ABB RAPID module: P90.mod

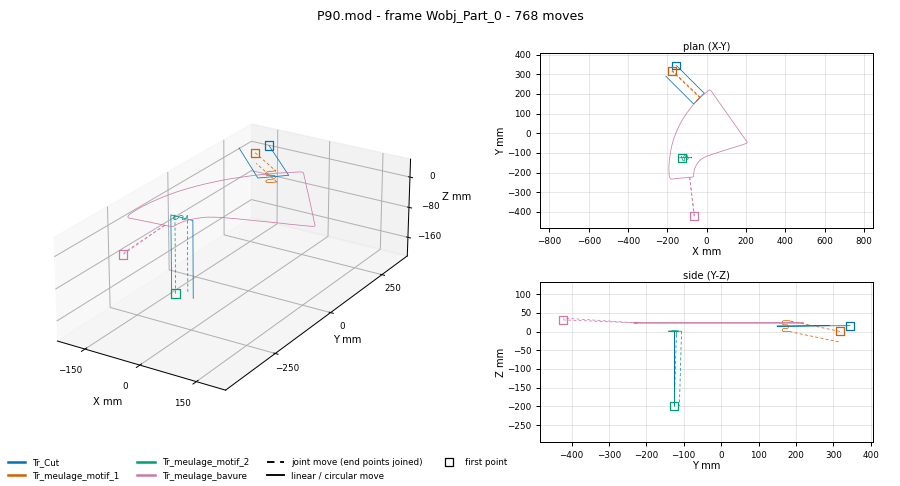
[picture p0: tool path of P90.mod in frame Wobj_Part_0, 768 of 778 moves have a stored position in this frame; points joined in program order, loops and branches not executed]
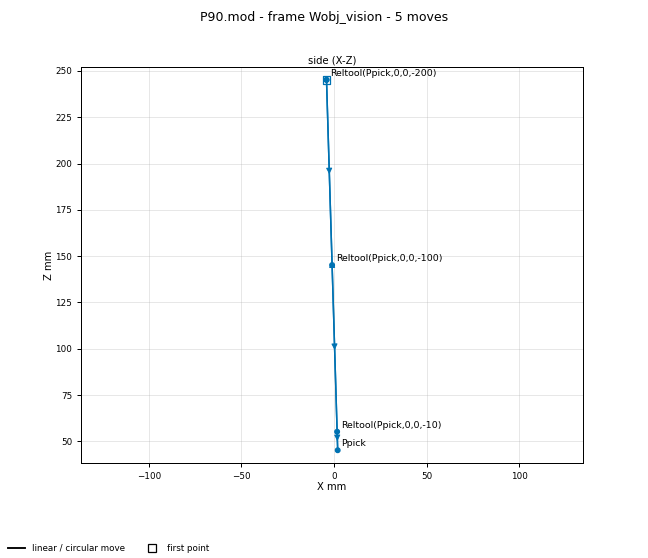
[picture p1: tool path of P90.mod in frame Wobj_vision, 5 of 778 moves have a stored position in this frame; points joined in program order, loops and branches not executed]
MODULE P90
	LOCAL CONST Speeddata vitesse_Tronconnage :=[10, 500, 0, 0];
	LOCAL CONST Robtarget Coupe_0 :=[[-42.54716015625,172.81159375,14.480369140625],[0.652659857981833,0.65438215651073,-0.267925350126422,-0.272093935579487],[0,0,0,0],[8.999999E+09,8.999999E+09,8.999999E+09,8.999999E+09,8.999999E+09,8.999999E+09]];
	LOCAL CONST Robtarget Coupe_1 :=[[-110.71790625,-124.2488046875,0.946675476074219],[0.708605063224334,-0.000599516120089683,-0.705604806156146,0.000602065284240644],[0,0,0,0],[8.999999E+09,8.999999E+09,8.999999E+09,8.999999E+09,8.999999E+09,8.999999E+09]];
	LOCAL CONST Robtarget Tr_meulage_motif_1_App1 :=[[-177.46862221102,317.614885440175,0.282455470844067],[0.29645362274748,-0.256571046125753,0.60201931555639,-0.695599950795604],[0,0,0,0],[8.999999E+09,8.999999E+09,8.999999E+09,8.999999E+09,8.999999E+09,8.999999E+09]];
	LOCAL CONST Robtarget Tr_meulage_motif_1_App2 :=[[-41.830808844926,187.387673178259,27.545191425886],[0.29645362274748,-0.256571046125753,0.60201931555639,-0.695599950795604],[0,0,0,0],[8.999999E+09,8.999999E+09,8.999999E+09,8.999999E+09,8.999999E+09,8.999999E+09]];
	LOCAL CONST Robtarget Tr_meulage_motif_1_P0 :=[[-34.6919765625,180.533609375,28.980072265625],[0.29645362274748,-0.256571046125753,0.60201931555639,-0.695599950795604],[0,0,0,0],[8.999999E+09,8.999999E+09,8.999999E+09,8.999999E+09,8.999999E+09,8.999999E+09]];
	LOCAL CONST Robtarget Tr_meulage_motif_1_P1 :=[[-35.39916796875,179.826578125,28.980072265625],[0.29645362274748,-0.256571046125753,0.60201931555639,-0.695599950795604],[0,0,0,0],[8.999999E+09,8.999999E+09,8.999999E+09,8.999999E+09,8.999999E+09,8.999999E+09]];
	LOCAL CONST Robtarget Tr_meulage_motif_1_P2 :=[[-36.106359375,179.1195625,28.980072265625],[0.29645362274748,-0.256571046125753,0.60201931555639,-0.695599950795604],[0,0,0,0],[8.999999E+09,8.999999E+09,8.999999E+09,8.999999E+09,8.999999E+09,8.999999E+09]];
	LOCAL CONST Robtarget Tr_meulage_motif_1_P3 :=[[-36.81355078125,178.41253125,28.980072265625],[0.29645362274748,-0.256571046125753,0.60201931555639,-0.695599950795604],[0,0,0,0],[8.999999E+09,8.999999E+09,8.999999E+09,8.999999E+09,8.999999E+09,8.999999E+09]];
	LOCAL CONST Robtarget Tr_meulage_motif_1_P4 :=[[-37.5207421875,177.705515625,28.980072265625],[0.29645362274748,-0.256571046125753,0.60201931555639,-0.695599950795604],[0,0,0,0],[8.999999E+09,8.999999E+09,8.999999E+09,8.999999E+09,8.999999E+09,8.999999E+09]];
	LOCAL CONST Robtarget Tr_meulage_motif_1_P5 :=[[-38.22793359375,176.9985,28.980072265625],[0.29645362274748,-0.256571046125753,0.60201931555639,-0.695599950795604],[0,0,0,0],[8.999999E+09,8.999999E+09,8.999999E+09,8.999999E+09,8.999999E+09,8.999999E+09]];
	LOCAL CONST Robtarget Tr_meulage_motif_1_P6 :=[[-38.935125,176.29146875,28.980072265625],[0.29645362274748,-0.256571046125753,0.60201931555639,-0.695599950795604],[0,0,0,0],[8.999999E+09,8.999999E+09,8.999999E+09,8.999999E+09,8.999999E+09,8.999999E+09]];
	LOCAL CONST Robtarget Tr_meulage_motif_1_P7 :=[[-39.64231640625,175.584453125,28.980072265625],[0.29645362274748,-0.256571046125753,0.60201931555639,-0.695599950795604],[0,0,0,0],[8.999999E+09,8.999999E+09,8.999999E+09,8.999999E+09,8.999999E+09,8.999999E+09]];
	LOCAL CONST Robtarget Tr_meulage_motif_1_P8 :=[[-40.3495078125,174.877421875,28.980072265625],[0.29645362274748,-0.256571046125753,0.60201931555639,-0.695599950795604],[0,0,0,0],[8.999999E+09,8.999999E+09,8.999999E+09,8.999999E+09,8.999999E+09,8.999999E+09]];
	LOCAL CONST Robtarget Tr_meulage_motif_1_P9 :=[[-41.05669921875,174.17040625,28.980072265625],[0.29645362274748,-0.256571046125753,0.60201931555639,-0.695599950795604],[0,0,0,0],[8.999999E+09,8.999999E+09,8.999999E+09,8.999999E+09,8.999999E+09,8.999999E+09]];
	LOCAL CONST Robtarget Tr_meulage_motif_1_P10 :=[[-41.76389453125,173.463390625,28.980072265625],[0.29645362274748,-0.256571046125753,0.60201931555639,-0.695599950795604],[0,0,0,0],[8.999999E+09,8.999999E+09,8.999999E+09,8.999999E+09,8.999999E+09,8.999999E+09]];
	LOCAL CONST Robtarget Tr_meulage_motif_1_P11 :=[[-42.4710859375,172.756359375,28.980072265625],[0.29645362274748,-0.256571046125753,0.60201931555639,-0.695599950795604],[0,0,0,0],[8.999999E+09,8.999999E+09,8.999999E+09,8.999999E+09,8.999999E+09,8.999999E+09]];
	LOCAL CONST Robtarget Tr_meulage_motif_1_P12 :=[[-43.17827734375,172.04934375,28.980072265625],[0.29645362274748,-0.256571046125753,0.60201931555639,-0.695599950795604],[0,0,0,0],[8.999999E+09,8.999999E+09,8.999999E+09,8.999999E+09,8.999999E+09,8.999999E+09]];
	LOCAL CONST Robtarget Tr_meulage_motif_1_P13 :=[[-43.88546875,171.3423125,28.980072265625],[0.29645362274748,-0.256571046125753,0.60201931555639,-0.695599950795604],[0,0,0,0],[8.999999E+09,8.999999E+09,8.999999E+09,8.999999E+09,8.999999E+09,8.999999E+09]];
	LOCAL CONST Robtarget Tr_meulage_motif_1_P14 :=[[-44.59266015625,170.635296875,28.980072265625],[0.29645362274748,-0.256571046125753,0.60201931555639,-0.695599950795604],[0,0,0,0],[8.999999E+09,8.999999E+09,8.999999E+09,8.999999E+09,8.999999E+09,8.999999E+09]];
	LOCAL CONST Robtarget Tr_meulage_motif_1_P15 :=[[-45.2998515625,169.92828125,28.980072265625],[0.29645362274748,-0.256571046125753,0.60201931555639,-0.695599950795604],[0,0,0,0],[8.999999E+09,8.999999E+09,8.999999E+09,8.999999E+09,8.999999E+09,8.999999E+09]];
	LOCAL CONST Robtarget Tr_meulage_motif_1_P16 :=[[-46.00704296875,169.22125,28.980072265625],[0.29645362274748,-0.256571046125753,0.60201931555639,-0.695599950795604],[0,0,0,0],[8.999999E+09,8.999999E+09,8.999999E+09,8.999999E+09,8.999999E+09,8.999999E+09]];
	LOCAL CONST Robtarget Tr_meulage_motif_1_P17 :=[[-46.714234375,168.514234375,28.980072265625],[0.29645362274748,-0.256571046125753,0.60201931555639,-0.695599950795604],[0,0,0,0],[8.999999E+09,8.999999E+09,8.999999E+09,8.999999E+09,8.999999E+09,8.999999E+09]];
	LOCAL CONST Robtarget Tr_meulage_motif_1_P18 :=[[-47.42142578125,167.807203125,28.980072265625],[0.29645362274748,-0.256571046125753,0.60201931555639,-0.695599950795604],[0,0,0,0],[8.999999E+09,8.999999E+09,8.999999E+09,8.999999E+09,8.999999E+09,8.999999E+09]];
	LOCAL CONST Robtarget Tr_meulage_motif_1_P19 :=[[-48.123859375,167.105953125,28.86948046875],[0.29645362274748,-0.256571046125753,0.60201931555639,-0.695599950795604],[0,0,0,0],[8.999999E+09,8.999999E+09,8.999999E+09,8.999999E+09,8.999999E+09,8.999999E+09]];
	LOCAL CONST Robtarget Tr_meulage_motif_1_P20 :=[[-48.794171875,166.437703125,28.658296875],[0.29645362274748,-0.256571046125753,0.60201931555639,-0.695599950795604],[0,0,0,0],[8.999999E+09,8.999999E+09,8.999999E+09,8.999999E+09,8.999999E+09,8.999999E+09]];
	LOCAL CONST Robtarget Tr_meulage_motif_1_P21 :=[[-49.3984375,165.836046875,28.386458984375],[0.29645362274748,-0.256571046125753,0.60201931555639,-0.695599950795604],[0,0,0,0],[8.999999E+09,8.999999E+09,8.999999E+09,8.999999E+09,8.999999E+09,8.999999E+09]];
	LOCAL CONST Robtarget Tr_meulage_motif_1_P22 :=[[-49.9300390625,165.307078125,28.11052734375],[0.29645362274748,-0.256571046125753,0.60201931555639,-0.695599950795604],[0,0,0,0],[8.999999E+09,8.999999E+09,8.999999E+09,8.999999E+09,8.999999E+09,8.999999E+09]];
	LOCAL CONST Robtarget Tr_meulage_motif_1_P23 :=[[-50.71148828125,164.531390625,27.494416015625],[0.29645362274748,-0.256571046125753,0.60201931555639,-0.695599950795604],[0,0,0,0],[8.999999E+09,8.999999E+09,8.999999E+09,8.999999E+09,8.999999E+09,8.999999E+09]];
	LOCAL CONST Robtarget Tr_meulage_motif_1_P24 :=[[-51.43940234375,163.811328125,26.64677734375],[0.29645362274748,-0.256571046125753,0.60201931555639,-0.695599950795604],[0,0,0,0],[8.999999E+09,8.999999E+09,8.999999E+09,8.999999E+09,8.999999E+09,8.999999E+09]];
	LOCAL CONST Robtarget Tr_meulage_motif_1_P25 :=[[-52.04349609375,163.21665625,25.622921875],[0.29645362274748,-0.256571046125753,0.60201931555639,-0.695599950795604],[0,0,0,0],[8.999999E+09,8.999999E+09,8.999999E+09,8.999999E+09,8.999999E+09,8.999999E+09]];
	LOCAL CONST Robtarget Tr_meulage_motif_1_P26 :=[[-52.393765625,162.8765625,24.5067578125],[0.29645362274748,-0.256571046125753,0.60201931555639,-0.695599950795604],[0,0,0,0],[8.999999E+09,8.999999E+09,8.999999E+09,8.999999E+09,8.999999E+09,8.999999E+09]];
	LOCAL CONST Robtarget Tr_meulage_motif_1_P27 :=[[-52.41605859375,162.86059375,23.810802734375],[0.29645362274748,-0.256571046125753,0.60201931555639,-0.695599950795604],[0,0,0,0],[8.999999E+09,8.999999E+09,8.999999E+09,8.999999E+09,8.999999E+09,8.999999E+09]];
	LOCAL CONST Robtarget Tr_meulage_motif_1_P28 :=[[-52.41905078125,162.863578125,23.14956640625],[0.29645362274748,-0.256571046125753,0.60201931555639,-0.695599950795604],[0,0,0,0],[8.999999E+09,8.999999E+09,8.999999E+09,8.999999E+09,8.999999E+09,8.999999E+09]];
	LOCAL CONST Robtarget Tr_meulage_motif_1_P29 :=[[-52.383234375,162.905375,22.488486328125],[0.29645362274748,-0.256571046125753,0.60201931555639,-0.695599950795604],[0,0,0,0],[8.999999E+09,8.999999E+09,8.999999E+09,8.999999E+09,8.999999E+09,8.999999E+09]];
	LOCAL CONST Robtarget Tr_meulage_motif_1_P30 :=[[-52.03588671875,163.262609375,21.386759765625],[0.29645362274748,-0.256571046125753,0.60201931555639,-0.695599950795604],[0,0,0,0],[8.999999E+09,8.999999E+09,8.999999E+09,8.999999E+09,8.999999E+09,8.999999E+09]];
	LOCAL CONST Robtarget Tr_meulage_motif_1_P31 :=[[-51.4346484375,163.872828125,20.380154296875],[0.29645362274748,-0.256571046125753,0.60201931555639,-0.695599950795604],[0,0,0,0],[8.999999E+09,8.999999E+09,8.999999E+09,8.999999E+09,8.999999E+09,8.999999E+09]];
	LOCAL CONST Robtarget Tr_meulage_motif_1_P32 :=[[-50.71465625,164.600140625,19.551296875],[0.29645362274748,-0.256571046125753,0.60201931555639,-0.695599950795604],[0,0,0,0],[8.999999E+09,8.999999E+09,8.999999E+09,8.999999E+09,8.999999E+09,8.999999E+09]];
	LOCAL CONST Robtarget Tr_meulage_motif_1_P33 :=[[-50.2305390625,165.087734375,19.1555546875],[0.29645362274748,-0.256571046125753,0.60201931555639,-0.695599950795604],[0,0,0,0],[8.999999E+09,8.999999E+09,8.999999E+09,8.999999E+09,8.999999E+09,8.999999E+09]];
	LOCAL CONST Robtarget Tr_meulage_motif_1_P34 :=[[-49.41370703125,165.90878125,18.668033203125],[0.29645362274748,-0.256571046125753,0.60201931555639,-0.695599950795604],[0,0,0,0],[8.999999E+09,8.999999E+09,8.999999E+09,8.999999E+09,8.999999E+09,8.999999E+09]];
	LOCAL CONST Robtarget Tr_meulage_motif_1_P35 :=[[-48.8173046875,166.5074375,18.4039453125],[0.29645362274748,-0.256571046125753,0.60201931555639,-0.695599950795604],[0,0,0,0],[8.999999E+09,8.999999E+09,8.999999E+09,8.999999E+09,8.999999E+09,8.999999E+09]];
	LOCAL CONST Robtarget Tr_meulage_motif_1_P36 :=[[-48.15912890625,167.167296875,18.19948046875],[0.29645362274748,-0.256571046125753,0.60201931555639,-0.695599950795604],[0,0,0,0],[8.999999E+09,8.999999E+09,8.999999E+09,8.999999E+09,8.999999E+09,8.999999E+09]];
	LOCAL CONST Robtarget Tr_meulage_motif_1_P37 :=[[-47.46546484375,167.86178125,18.090888671875],[0.29645362274748,-0.256571046125753,0.60201931555639,-0.695599950795604],[0,0,0,0],[8.999999E+09,8.999999E+09,8.999999E+09,8.999999E+09,8.999999E+09,8.999999E+09]];
	LOCAL CONST Robtarget Tr_meulage_motif_1_P38 :=[[-46.76403515625,168.564046875,17.980296875],[0.29645362274748,-0.256571046125753,0.60201931555639,-0.695599950795604],[0,0,0,0],[8.999999E+09,8.999999E+09,8.999999E+09,8.999999E+09,8.999999E+09,8.999999E+09]];
	LOCAL CONST Robtarget Tr_meulage_motif_1_P39 :=[[-46.05684375,169.2710625,17.980296875],[0.29645362274748,-0.256571046125753,0.60201931555639,-0.695599950795604],[0,0,0,0],[8.999999E+09,8.999999E+09,8.999999E+09,8.999999E+09,8.999999E+09,8.999999E+09]];
	LOCAL CONST Robtarget Tr_meulage_motif_1_P40 :=[[-45.34965234375,169.97809375,17.980296875],[0.29645362274748,-0.256571046125753,0.60201931555639,-0.695599950795604],[0,0,0,0],[8.999999E+09,8.999999E+09,8.999999E+09,8.999999E+09,8.999999E+09,8.999999E+09]];
	LOCAL CONST Robtarget Tr_meulage_motif_1_P41 :=[[-44.6424609375,170.685109375,17.980296875],[0.29645362274748,-0.256571046125753,0.60201931555639,-0.695599950795604],[0,0,0,0],[8.999999E+09,8.999999E+09,8.999999E+09,8.999999E+09,8.999999E+09,8.999999E+09]];
	LOCAL CONST Robtarget Tr_meulage_motif_1_P42 :=[[-43.935265625,171.392125,17.980296875],[0.29645362274748,-0.256571046125753,0.60201931555639,-0.695599950795604],[0,0,0,0],[8.999999E+09,8.999999E+09,8.999999E+09,8.999999E+09,8.999999E+09,8.999999E+09]];
	LOCAL CONST Robtarget Tr_meulage_motif_1_P43 :=[[-43.22807421875,172.09915625,17.980296875],[0.29645362274748,-0.256571046125753,0.60201931555639,-0.695599950795604],[0,0,0,0],[8.999999E+09,8.999999E+09,8.999999E+09,8.999999E+09,8.999999E+09,8.999999E+09]];
	LOCAL CONST Robtarget Tr_meulage_motif_1_P44 :=[[-42.5208828125,172.806171875,17.980296875],[0.29645362274748,-0.256571046125753,0.60201931555639,-0.695599950795604],[0,0,0,0],[8.999999E+09,8.999999E+09,8.999999E+09,8.999999E+09,8.999999E+09,8.999999E+09]];
	LOCAL CONST Robtarget Tr_meulage_motif_1_P45 :=[[-41.81369140625,173.5131875,17.980296875],[0.29645362274748,-0.256571046125753,0.60201931555639,-0.695599950795604],[0,0,0,0],[8.999999E+09,8.999999E+09,8.999999E+09,8.999999E+09,8.999999E+09,8.999999E+09]];
	LOCAL CONST Robtarget Tr_meulage_motif_1_P46 :=[[-41.1065,174.22021875,17.980296875],[0.29645362274748,-0.256571046125753,0.60201931555639,-0.695599950795604],[0,0,0,0],[8.999999E+09,8.999999E+09,8.999999E+09,8.999999E+09,8.999999E+09,8.999999E+09]];
	LOCAL CONST Robtarget Tr_meulage_motif_1_P47 :=[[-40.39930859375,174.927234375,17.980296875],[0.29645362274748,-0.256571046125753,0.60201931555639,-0.695599950795604],[0,0,0,0],[8.999999E+09,8.999999E+09,8.999999E+09,8.999999E+09,8.999999E+09,8.999999E+09]];
	LOCAL CONST Robtarget Tr_meulage_motif_1_P48 :=[[-39.6921171875,175.634265625,17.980296875],[0.29645362274748,-0.256571046125753,0.60201931555639,-0.695599950795604],[0,0,0,0],[8.999999E+09,8.999999E+09,8.999999E+09,8.999999E+09,8.999999E+09,8.999999E+09]];
	LOCAL CONST Robtarget Tr_meulage_motif_1_P49 :=[[-38.99068359375,176.33653125,17.869705078125],[0.29645362274748,-0.256571046125753,0.60201931555639,-0.695599950795604],[0,0,0,0],[8.999999E+09,8.999999E+09,8.999999E+09,8.999999E+09,8.999999E+09,8.999999E+09]];
	LOCAL CONST Robtarget Tr_meulage_motif_1_P50 :=[[-38.32228515625,177.006671875,17.6585234375],[0.29645362274748,-0.256571046125753,0.60201931555639,-0.695599950795604],[0,0,0,0],[8.999999E+09,8.999999E+09,8.999999E+09,8.999999E+09,8.999999E+09,8.999999E+09]];
	LOCAL CONST Robtarget Tr_meulage_motif_1_P51 :=[[-37.72048046875,177.610796875,17.38668359375],[0.29645362274748,-0.256571046125753,0.60201931555639,-0.695599950795604],[0,0,0,0],[8.999999E+09,8.999999E+09,8.999999E+09,8.999999E+09,8.999999E+09,8.999999E+09]];
	LOCAL CONST Robtarget Tr_meulage_motif_1_P52 :=[[-37.2186875,178.11521875,17.08253515625],[0.29645362274748,-0.256571046125753,0.60201931555639,-0.695599950795604],[0,0,0,0],[8.999999E+09,8.999999E+09,8.999999E+09,8.999999E+09,8.999999E+09,8.999999E+09]];
	LOCAL CONST Robtarget Tr_meulage_motif_1_P53 :=[[-36.49012109375,178.849609375,16.420015625],[0.29645362274748,-0.256571046125753,0.60201931555639,-0.695599950795604],[0,0,0,0],[8.999999E+09,8.999999E+09,8.999999E+09,8.999999E+09,8.999999E+09,8.999999E+09]];
	LOCAL CONST Robtarget Tr_meulage_motif_1_P54 :=[[-35.85636328125,179.491390625,15.51809765625],[0.29645362274748,-0.256571046125753,0.60201931555639,-0.695599950795604],[0,0,0,0],[8.999999E+09,8.999999E+09,8.999999E+09,8.999999E+09,8.999999E+09,8.999999E+09]];
	LOCAL CONST Robtarget Tr_meulage_motif_1_P55 :=[[-35.4827734375,179.874359375,14.472087890625],[0.29645362274748,-0.256571046125753,0.60201931555639,-0.695599950795604],[0,0,0,0],[8.999999E+09,8.999999E+09,8.999999E+09,8.999999E+09,8.999999E+09,8.999999E+09]];
	LOCAL CONST Robtarget Tr_meulage_motif_1_P56 :=[[-35.355234375,180.008140625,13.7788828125],[0.29645362274748,-0.256571046125753,0.60201931555639,-0.695599950795604],[0,0,0,0],[8.999999E+09,8.999999E+09,8.999999E+09,8.999999E+09,8.999999E+09,8.999999E+09]];
	LOCAL CONST Robtarget Tr_meulage_motif_1_P57 :=[[-35.3135703125,180.056765625,13.0088984375],[0.29645362274748,-0.256571046125753,0.60201931555639,-0.695599950795604],[0,0,0,0],[8.999999E+09,8.999999E+09,8.999999E+09,8.999999E+09,8.999999E+09,8.999999E+09]];
	LOCAL CONST Robtarget Tr_meulage_motif_1_P58 :=[[-35.36439453125,180.012921875,12.2390400390625],[0.29645362274748,-0.256571046125753,0.60201931555639,-0.695599950795604],[0,0,0,0],[8.999999E+09,8.999999E+09,8.999999E+09,8.999999E+09,8.999999E+09,8.999999E+09]];
	LOCAL CONST Robtarget Tr_meulage_motif_1_P59 :=[[-35.66614453125,179.72128125,11.1308125],[0.29645362274748,-0.256571046125753,0.60201931555639,-0.695599950795604],[0,0,0,0],[8.999999E+09,8.999999E+09,8.999999E+09,8.999999E+09,8.999999E+09,8.999999E+09]];
	LOCAL CONST Robtarget Tr_meulage_motif_1_P60 :=[[-35.96179296875,179.431015625,10.54513671875],[0.29645362274748,-0.256571046125753,0.60201931555639,-0.695599950795604],[0,0,0,0],[8.999999E+09,8.999999E+09,8.999999E+09,8.999999E+09,8.999999E+09,8.999999E+09]];
	LOCAL CONST Robtarget Tr_meulage_motif_1_P61 :=[[-36.59317578125,178.8078125,9.6580302734375],[0.29645362274748,-0.256571046125753,0.60201931555639,-0.695599950795604],[0,0,0,0],[8.999999E+09,8.999999E+09,8.999999E+09,8.999999E+09,8.999999E+09,8.999999E+09]];
	LOCAL CONST Robtarget Tr_meulage_motif_1_P62 :=[[-37.00924609375,178.39559375,9.2437265625],[0.29645362274748,-0.256571046125753,0.60201931555639,-0.695599950795604],[0,0,0,0],[8.999999E+09,8.999999E+09,8.999999E+09,8.999999E+09,8.999999E+09,8.999999E+09]];
	LOCAL CONST Robtarget Tr_meulage_motif_1_P63 :=[[-37.80228515625,177.607671875,8.6996435546875],[0.29645362274748,-0.256571046125753,0.60201931555639,-0.695599950795604],[0,0,0,0],[8.999999E+09,8.999999E+09,8.999999E+09,8.999999E+09,8.999999E+09,8.999999E+09]];
	LOCAL CONST Robtarget Tr_meulage_motif_1_P64 :=[[-38.3874765625,177.025296875,8.4041494140625],[0.29645362274748,-0.256571046125753,0.60201931555639,-0.695599950795604],[0,0,0,0],[8.999999E+09,8.999999E+09,8.999999E+09,8.999999E+09,8.999999E+09,8.999999E+09]];
	LOCAL CONST Robtarget Tr_meulage_motif_1_P65 :=[[-39.04750390625,176.36728125,8.199685546875],[0.29645362274748,-0.256571046125753,0.60201931555639,-0.695599950795604],[0,0,0,0],[8.999999E+09,8.999999E+09,8.999999E+09,8.999999E+09,8.999999E+09,8.999999E+09]];
	LOCAL CONST Robtarget Tr_meulage_motif_1_P66 :=[[-39.7421484375,175.67378125,8.09109375],[0.29645362274748,-0.256571046125753,0.60201931555639,-0.695599950795604],[0,0,0,0],[8.999999E+09,8.999999E+09,8.999999E+09,8.999999E+09,8.999999E+09,8.999999E+09]];
	LOCAL CONST Robtarget Tr_meulage_motif_1_P67 :=[[-40.44458203125,174.972515625,7.98050244140625],[0.29645362274748,-0.256571046125753,0.60201931555639,-0.695599950795604],[0,0,0,0],[8.999999E+09,8.999999E+09,8.999999E+09,8.999999E+09,8.999999E+09,8.999999E+09]];
	LOCAL CONST Robtarget Tr_meulage_motif_1_P68 :=[[-41.1517734375,174.2655,7.98050244140625],[0.29645362274748,-0.256571046125753,0.60201931555639,-0.695599950795604],[0,0,0,0],[8.999999E+09,8.999999E+09,8.999999E+09,8.999999E+09,8.999999E+09,8.999999E+09]];
	LOCAL CONST Robtarget Tr_meulage_motif_1_P69 :=[[-41.85896484375,173.558484375,7.98050244140625],[0.29645362274748,-0.256571046125753,0.60201931555639,-0.695599950795604],[0,0,0,0],[8.999999E+09,8.999999E+09,8.999999E+09,8.999999E+09,8.999999E+09,8.999999E+09]];
	LOCAL CONST Robtarget Tr_meulage_motif_1_P70 :=[[-42.56615625,172.851453125,7.98050244140625],[0.29645362274748,-0.256571046125753,0.60201931555639,-0.695599950795604],[0,0,0,0],[8.999999E+09,8.999999E+09,8.999999E+09,8.999999E+09,8.999999E+09,8.999999E+09]];
	LOCAL CONST Robtarget Tr_meulage_motif_1_P71 :=[[-43.27334765625,172.1444375,7.98050244140625],[0.29645362274748,-0.256571046125753,0.60201931555639,-0.695599950795604],[0,0,0,0],[8.999999E+09,8.999999E+09,8.999999E+09,8.999999E+09,8.999999E+09,8.999999E+09]];
	LOCAL CONST Robtarget Tr_meulage_motif_1_P72 :=[[-43.9805390625,171.43740625,7.98050244140625],[0.29645362274748,-0.256571046125753,0.60201931555639,-0.695599950795604],[0,0,0,0],[8.999999E+09,8.999999E+09,8.999999E+09,8.999999E+09,8.999999E+09,8.999999E+09]];
	LOCAL CONST Robtarget Tr_meulage_motif_1_P73 :=[[-44.68773046875,170.730390625,7.98050244140625],[0.29645362274748,-0.256571046125753,0.60201931555639,-0.695599950795604],[0,0,0,0],[8.999999E+09,8.999999E+09,8.999999E+09,8.999999E+09,8.999999E+09,8.999999E+09]];
	LOCAL CONST Robtarget Tr_meulage_motif_1_P74 :=[[-45.394921875,170.023375,7.98050244140625],[0.29645362274748,-0.256571046125753,0.60201931555639,-0.695599950795604],[0,0,0,0],[8.999999E+09,8.999999E+09,8.999999E+09,8.999999E+09,8.999999E+09,8.999999E+09]];
	LOCAL CONST Robtarget Tr_meulage_motif_1_P75 :=[[-46.10211328125,169.31634375,7.98050244140625],[0.29645362274748,-0.256571046125753,0.60201931555639,-0.695599950795604],[0,0,0,0],[8.999999E+09,8.999999E+09,8.999999E+09,8.999999E+09,8.999999E+09,8.999999E+09]];
	LOCAL CONST Robtarget Tr_meulage_motif_1_P76 :=[[-46.80930859375,168.609328125,7.98050244140625],[0.29645362274748,-0.256571046125753,0.60201931555639,-0.695599950795604],[0,0,0,0],[8.999999E+09,8.999999E+09,8.999999E+09,8.999999E+09,8.999999E+09,8.999999E+09]];
	LOCAL CONST Robtarget Tr_meulage_motif_1_P77 :=[[-47.5165,167.902296875,7.9805029296875],[0.29645362274748,-0.256571046125753,0.60201931555639,-0.695599950795604],[0,0,0,0],[8.999999E+09,8.999999E+09,8.999999E+09,8.999999E+09,8.999999E+09,8.999999E+09]];
	LOCAL CONST Robtarget Tr_meulage_motif_1_P78 :=[[-48.2189296875,167.201046875,7.8699111328125],[0.29645362274748,-0.256571046125753,0.60201931555639,-0.695599950795604],[0,0,0,0],[8.999999E+09,8.999999E+09,8.999999E+09,8.999999E+09,8.999999E+09,8.999999E+09]];
	LOCAL CONST Robtarget Tr_meulage_motif_1_P79 :=[[-48.88924609375,166.532796875,7.65872802734375],[0.29645362274748,-0.256571046125753,0.60201931555639,-0.695599950795604],[0,0,0,0],[8.999999E+09,8.999999E+09,8.999999E+09,8.999999E+09,8.999999E+09,8.999999E+09]];
	LOCAL CONST Robtarget Tr_meulage_motif_1_P80 :=[[-49.49351171875,165.931140625,7.38689013671875],[0.29645362274748,-0.256571046125753,0.60201931555639,-0.695599950795604],[0,0,0,0],[8.999999E+09,8.999999E+09,8.999999E+09,8.999999E+09,8.999999E+09,8.999999E+09]];
	LOCAL CONST Robtarget Tr_meulage_motif_1_P81 :=[[-50.025109375,165.402171875,7.1109580078125],[0.29645362274748,-0.256571046125753,0.60201931555639,-0.695599950795604],[0,0,0,0],[8.999999E+09,8.999999E+09,8.999999E+09,8.999999E+09,8.999999E+09,8.999999E+09]];
	LOCAL CONST Robtarget Tr_meulage_motif_1_P82 :=[[-50.8065625,164.626484375,6.494845703125],[0.29645362274748,-0.256571046125753,0.60201931555639,-0.695599950795604],[0,0,0,0],[8.999999E+09,8.999999E+09,8.999999E+09,8.999999E+09,8.999999E+09,8.999999E+09]];
	LOCAL CONST Robtarget Tr_meulage_motif_1_P83 :=[[-51.48719140625,163.954109375,5.6008955078125],[0.29645362274748,-0.256571046125753,0.60201931555639,-0.695599950795604],[0,0,0,0],[8.999999E+09,8.999999E+09,8.999999E+09,8.999999E+09,8.999999E+09,8.999999E+09]];
	LOCAL CONST Robtarget Tr_meulage_motif_1_P84 :=[[-51.92287890625,163.528359375,4.51491796875],[0.29645362274748,-0.256571046125753,0.60201931555639,-0.695599950795604],[0,0,0,0],[8.999999E+09,8.999999E+09,8.999999E+09,8.999999E+09,8.999999E+09,8.999999E+09]];
	LOCAL CONST Robtarget Tr_meulage_motif_1_P85 :=[[-52.0470703125,163.413109375,3.53056298828125],[0.29645362274748,-0.256571046125753,0.60201931555639,-0.695599950795604],[0,0,0,0],[8.999999E+09,8.999999E+09,8.999999E+09,8.999999E+09,8.999999E+09,8.999999E+09]];
	LOCAL CONST Robtarget Tr_meulage_motif_1_P86 :=[[-51.9550234375,163.506984375,3.32591088867188],[0.29645362274748,-0.256571046125753,0.60201931555639,-0.695599950795604],[0,0,0,0],[8.999999E+09,8.999999E+09,8.999999E+09,8.999999E+09,8.999999E+09,8.999999E+09]];
	LOCAL CONST Robtarget Tr_meulage_motif_1_P87 :=[[-51.8710625,163.597515625,2.59951953125],[0.29645362274748,-0.256571046125753,0.60201931555639,-0.695599950795604],[0,0,0,0],[8.999999E+09,8.999999E+09,8.999999E+09,8.999999E+09,8.999999E+09,8.999999E+09]];
	LOCAL CONST Robtarget Tr_meulage_motif_1_P88 :=[[-51.3915859375,164.085359375,1.66263244628906],[0.29645362274748,-0.256571046125753,0.60201931555639,-0.695599950795604],[0,0,0,0],[8.999999E+09,8.999999E+09,8.999999E+09,8.999999E+09,8.999999E+09,8.999999E+09]];
	LOCAL CONST Robtarget Tr_meulage_motif_1_P89 :=[[-50.9993359375,164.481703125,1.19882946777344],[0.29645362274748,-0.256571046125753,0.60201931555639,-0.695599950795604],[0,0,0,0],[8.999999E+09,8.999999E+09,8.999999E+09,8.999999E+09,8.999999E+09,8.999999E+09]];
	LOCAL CONST Robtarget Tr_meulage_motif_1_P90 :=[[-50.202390625,165.283265625,0.668402770996094],[0.29645362274748,-0.256571046125753,0.60201931555639,-0.695599950795604],[0,0,0,0],[8.999999E+09,8.999999E+09,8.999999E+09,8.999999E+09,8.999999E+09,8.999999E+09]];
	LOCAL CONST Robtarget Tr_meulage_motif_1_P91 :=[[-49.605984375,165.881921875,0.404314422607422],[0.29645362274748,-0.256571046125753,0.60201931555639,-0.695599950795604],[0,0,0,0],[8.999999E+09,8.999999E+09,8.999999E+09,8.999999E+09,8.999999E+09,8.999999E+09]];
	LOCAL CONST Robtarget Tr_meulage_motif_1_P92 :=[[-48.94780859375,166.54178125,0.199849807739258],[0.29645362274748,-0.256571046125753,0.60201931555639,-0.695599950795604],[0,0,0,0],[8.999999E+09,8.999999E+09,8.999999E+09,8.999999E+09,8.999999E+09,8.999999E+09]];
	LOCAL CONST Robtarget Tr_meulage_motif_1_P93 :=[[-48.2541484375,167.236265625,0.0912582397460937],[0.29645362274748,-0.256571046125753,0.60201931555639,-0.695599950795604],[0,0,0,0],[8.999999E+09,8.999999E+09,8.999999E+09,8.999999E+09,8.999999E+09,8.999999E+09]];
	LOCAL CONST Robtarget Tr_meulage_motif_1_P94 :=[[-47.55271484375,167.93853125,-0.0193332862854004],[0.29645362274748,-0.256571046125753,0.60201931555639,-0.695599950795604],[0,0,0,0],[8.999999E+09,8.999999E+09,8.999999E+09,8.999999E+09,8.999999E+09,8.999999E+09]];
	LOCAL CONST Robtarget Tr_meulage_motif_1_P95 :=[[-46.8455234375,168.645546875,-0.0193333320617676],[0.29645362274748,-0.256571046125753,0.60201931555639,-0.695599950795604],[0,0,0,0],[8.999999E+09,8.999999E+09,8.999999E+09,8.999999E+09,8.999999E+09,8.999999E+09]];
	LOCAL CONST Robtarget Tr_meulage_motif_1_P96 :=[[-46.13833203125,169.352578125,-0.0193333759307861],[0.29645362274748,-0.256571046125753,0.60201931555639,-0.695599950795604],[0,0,0,0],[8.999999E+09,8.999999E+09,8.999999E+09,8.999999E+09,8.999999E+09,8.999999E+09]];
	LOCAL CONST Robtarget Tr_meulage_motif_1_P97 :=[[-45.431140625,170.05959375,-0.0193334217071533],[0.29645362274748,-0.256571046125753,0.60201931555639,-0.695599950795604],[0,0,0,0],[8.999999E+09,8.999999E+09,8.999999E+09,8.999999E+09,8.999999E+09,8.999999E+09]];
	LOCAL CONST Robtarget Tr_meulage_motif_1_P98 :=[[-44.72394921875,170.766609375,-0.0193334674835205],[0.29645362274748,-0.256571046125753,0.60201931555639,-0.695599950795604],[0,0,0,0],[8.999999E+09,8.999999E+09,8.999999E+09,8.999999E+09,8.999999E+09,8.999999E+09]];
	LOCAL CONST Robtarget Tr_meulage_motif_1_P99 :=[[-44.0167578125,171.473640625,-0.0193335113525391],[0.29645362274748,-0.256571046125753,0.60201931555639,-0.695599950795604],[0,0,0,0],[8.999999E+09,8.999999E+09,8.999999E+09,8.999999E+09,8.999999E+09,8.999999E+09]];
	LOCAL CONST Robtarget Tr_meulage_motif_1_P100 :=[[-43.30956640625,172.18065625,-0.0193335571289063],[0.29645362274748,-0.256571046125753,0.60201931555639,-0.695599950795604],[0,0,0,0],[8.999999E+09,8.999999E+09,8.999999E+09,8.999999E+09,8.999999E+09,8.999999E+09]];
	LOCAL CONST Robtarget Tr_meulage_motif_1_P101 :=[[-42.602375,172.8876875,-0.0193336009979248],[0.29645362274748,-0.256571046125753,0.60201931555639,-0.695599950795604],[0,0,0,0],[8.999999E+09,8.999999E+09,8.999999E+09,8.999999E+09,8.999999E+09,8.999999E+09]];
	LOCAL CONST Robtarget Tr_meulage_motif_1_P102 :=[[-41.89518359375,173.594703125,-0.019333646774292],[0.29645362274748,-0.256571046125753,0.60201931555639,-0.695599950795604],[0,0,0,0],[8.999999E+09,8.999999E+09,8.999999E+09,8.999999E+09,8.999999E+09,8.999999E+09]];
	LOCAL CONST Robtarget Tr_meulage_motif_1_P103 :=[[-41.18798828125,174.30171875,-0.0193336925506592],[0.29645362274748,-0.256571046125753,0.60201931555639,-0.695599950795604],[0,0,0,0],[8.999999E+09,8.999999E+09,8.999999E+09,8.999999E+09,8.999999E+09,8.999999E+09]];
	LOCAL CONST Robtarget Tr_meulage_motif_1_P104 :=[[-40.480796875,175.00875,-0.0193337364196777],[0.29645362274748,-0.256571046125753,0.60201931555639,-0.695599950795604],[0,0,0,0],[8.999999E+09,8.999999E+09,8.999999E+09,8.999999E+09,8.999999E+09,8.999999E+09]];
	LOCAL CONST Robtarget Tr_meulage_motif_1_P105 :=[[-39.77360546875,175.715765625,-0.0193337821960449],[0.29645362274748,-0.256571046125753,0.60201931555639,-0.695599950795604],[0,0,0,0],[8.999999E+09,8.999999E+09,8.999999E+09,8.999999E+09,8.999999E+09,8.999999E+09]];
	LOCAL CONST Robtarget Tr_meulage_motif_1_P106 :=[[-39.0664140625,176.422796875,-0.0193338279724121],[0.29645362274748,-0.256571046125753,0.60201931555639,-0.695599950795604],[0,0,0,0],[8.999999E+09,8.999999E+09,8.999999E+09,8.999999E+09,8.999999E+09,8.999999E+09]];
	LOCAL CONST Robtarget Tr_meulage_motif_1_P107 :=[[-38.35922265625,177.1298125,-0.0193338718414307],[0.29645362274748,-0.256571046125753,0.60201931555639,-0.695599950795604],[0,0,0,0],[8.999999E+09,8.999999E+09,8.999999E+09,8.999999E+09,8.999999E+09,8.999999E+09]];
	LOCAL CONST Robtarget Tr_meulage_motif_1_P108 :=[[-37.65203125,177.836828125,-0.0193339176177979],[0.29645362274748,-0.256571046125753,0.60201931555639,-0.695599950795604],[0,0,0,0],[8.999999E+09,8.999999E+09,8.999999E+09,8.999999E+09,8.999999E+09,8.999999E+09]];
	LOCAL CONST Robtarget Tr_meulage_motif_1_P109 :=[[-36.94483984375,178.543859375,-0.0193339614868164],[0.29645362274748,-0.256571046125753,0.60201931555639,-0.695599950795604],[0,0,0,0],[8.999999E+09,8.999999E+09,8.999999E+09,8.999999E+09,8.999999E+09,8.999999E+09]];
	LOCAL CONST Robtarget Tr_meulage_motif_1_P110 :=[[-36.2376484375,179.250875,-0.0193340072631836],[0.29645362274748,-0.256571046125753,0.60201931555639,-0.695599950795604],[0,0,0,0],[8.999999E+09,8.999999E+09,8.999999E+09,8.999999E+09,8.999999E+09,8.999999E+09]];
	LOCAL CONST Robtarget Tr_meulage_motif_1_P111 :=[[-35.53045703125,179.95790625,-0.0193340530395508],[0.29645362274748,-0.256571046125753,0.60201931555639,-0.695599950795604],[0,0,0,0],[8.999999E+09,8.999999E+09,8.999999E+09,8.999999E+09,8.999999E+09,8.999999E+09]];
	LOCAL CONST Robtarget Tr_meulage_motif_1_P112 :=[[-34.823265625,180.664921875,-0.0193340969085693],[0.29645362274748,-0.256571046125753,0.60201931555639,-0.695599950795604],[0,0,0,0],[8.999999E+09,8.999999E+09,8.999999E+09,8.999999E+09,8.999999E+09,8.999999E+09]];
	LOCAL CONST Robtarget Tr_meulage_motif_1_P113 :=[[-34.1160703125,181.3719375,-0.0193341426849365],[0.29645362274748,-0.256571046125753,0.60201931555639,-0.695599950795604],[0,0,0,0],[8.999999E+09,8.999999E+09,8.999999E+09,8.999999E+09,8.999999E+09,8.999999E+09]];
	LOCAL CONST Robtarget Tr_meulage_motif_1_P114 :=[[-33.40887890625,182.07896875,-0.0193341865539551],[0.29645362274748,-0.256571046125753,0.60201931555639,-0.695599950795604],[0,0,0,0],[8.999999E+09,8.999999E+09,8.999999E+09,8.999999E+09,8.999999E+09,8.999999E+09]];
	LOCAL CONST Robtarget Tr_meulage_motif_1_P115 :=[[-32.701689453125,182.785984375,-0.0193342323303223],[0.29645362274748,-0.256571046125753,0.60201931555639,-0.695599950795604],[0,0,0,0],[8.999999E+09,8.999999E+09,8.999999E+09,8.999999E+09,8.999999E+09,8.999999E+09]];
	LOCAL CONST Robtarget Tr_meulage_motif_1_degg1 :=[[-39.840521735551,189.640048178259,-1.45421507206937],[0.29645362274748,-0.256571046125753,0.60201931555639,-0.695599950795604],[0,0,0,0],[8.999999E+09,8.999999E+09,8.999999E+09,8.999999E+09,8.999999E+09,8.999999E+09]];
	LOCAL CONST Robtarget Tr_meulage_motif_1_degg2 :=[[-175.478335101645,319.867260440175,-28.7169510271113],[0.29645362274748,-0.256571046125753,0.60201931555639,-0.695599950795604],[0,0,0,0],[8.999999E+09,8.999999E+09,8.999999E+09,8.999999E+09,8.999999E+09,8.999999E+09]];
	LOCAL CONST Robtarget Tr_meulage_motif_2_App1 :=[[-125.376179622768,-125.082076727597,-198.959840528543],[-0.000102703814941082,0.00724489345550854,-0.0141742320669124,-0.999873288030067],[0,0,0,0],[8.999999E+09,8.999999E+09,8.999999E+09,8.999999E+09,8.999999E+09,8.999999E+09]];
	LOCAL CONST Robtarget Tr_meulage_motif_2_App2 :=[[-128.128337106138,-119.696268289505,-9.05613151617326],[-0.000102703814941082,0.00724489345550854,-0.0141742320669124,-0.999873288030067],[0,0,0,0],[8.999999E+09,8.999999E+09,8.999999E+09,8.999999E+09,8.999999E+09,8.999999E+09]];
	LOCAL CONST Robtarget Tr_meulage_motif_2_P0 :=[[-128.2731875,-119.4128046875,0.938800537109375],[-0.000102703814941082,0.00724489345550854,-0.0141742320669124,-0.999873288030067],[0,0,0,0],[8.999999E+09,8.999999E+09,8.999999E+09,8.999999E+09,8.999999E+09,8.999999E+09]];
	LOCAL CONST Robtarget Tr_meulage_motif_2_P1 :=[[-127.9014921875,-120.3411640625,0.940370422363281],[-0.000102703814941082,0.00724489345550854,-0.0141742320669124,-0.999873288030067],[0,0,0,0],[8.999999E+09,8.999999E+09,8.999999E+09,8.999999E+09,8.999999E+09,8.999999E+09]];
	LOCAL CONST Robtarget Tr_meulage_motif_2_P2 :=[[-127.5297890625,-121.269515625,0.941940307617188],[-0.000102703814941082,0.00724489345550854,-0.0141742320669124,-0.999873288030067],[0,0,0,0],[8.999999E+09,8.999999E+09,8.999999E+09,8.999999E+09,8.999999E+09,8.999999E+09]];
	LOCAL CONST Robtarget Tr_meulage_motif_2_P3 :=[[-127.15809375,-122.1978671875,0.943510192871094],[-0.000102703814941082,0.00724489345550854,-0.0141742320669124,-0.999873288030067],[0,0,0,0],[8.999999E+09,8.999999E+09,8.999999E+09,8.999999E+09,8.999999E+09,8.999999E+09]];
	LOCAL CONST Robtarget Tr_meulage_motif_2_P4 :=[[-126.7863984375,-123.12621875,0.945080078125],[-0.000102703814941082,0.00724489345550854,-0.0141742320669124,-0.999873288030067],[0,0,0,0],[8.999999E+09,8.999999E+09,8.999999E+09,8.999999E+09,8.999999E+09,8.999999E+09]];
	LOCAL CONST Robtarget Tr_meulage_motif_2_P5 :=[[-126.414703125,-124.0545703125,0.946649963378906],[-0.000102703814941082,0.00724489345550854,-0.0141742320669124,-0.999873288030067],[0,0,0,0],[8.999999E+09,8.999999E+09,8.999999E+09,8.999999E+09,8.999999E+09,8.999999E+09]];
	LOCAL CONST Robtarget Tr_meulage_motif_2_P6 :=[[-126.0430078125,-124.9829296875,0.948219848632813],[-0.000102703814941082,0.00724489345550854,-0.0141742320669124,-0.999873288030067],[0,0,0,0],[8.999999E+09,8.999999E+09,8.999999E+09,8.999999E+09,8.999999E+09,8.999999E+09]];
	LOCAL CONST Robtarget Tr_meulage_motif_2_P7 :=[[-125.6713125,-125.91128125,0.949789733886719],[-0.000102703814941082,0.00724489345550854,-0.0141742320669124,-0.999873288030067],[0,0,0,0],[8.999999E+09,8.999999E+09,8.999999E+09,8.999999E+09,8.999999E+09,8.999999E+09]];
	LOCAL CONST Robtarget Tr_meulage_motif_2_P8 :=[[-125.2996171875,-126.8396328125,0.951359680175781],[-0.000102703814941082,0.00724489345550854,-0.0141742320669124,-0.999873288030067],[0,0,0,0],[8.999999E+09,8.999999E+09,8.999999E+09,8.999999E+09,8.999999E+09,8.999999E+09]];
	LOCAL CONST Robtarget Tr_meulage_motif_2_P9 :=[[-124.927921875,-127.767984375,0.952929565429688],[-0.000102703814941082,0.00724489345550854,-0.0141742320669124,-0.999873288030067],[0,0,0,0],[8.999999E+09,8.999999E+09,8.999999E+09,8.999999E+09,8.999999E+09,8.999999E+09]];
	LOCAL CONST Robtarget Tr_meulage_motif_2_P10 :=[[-124.5562265625,-128.69634375,0.954499450683594],[-0.000102703814941082,0.00724489345550854,-0.0141742320669124,-0.999873288030067],[0,0,0,0],[8.999999E+09,8.999999E+09,8.999999E+09,8.999999E+09,8.999999E+09,8.999999E+09]];
	LOCAL CONST Robtarget Tr_meulage_motif_2_P11 :=[[-124.18453125,-129.6246953125,0.9560693359375],[-0.000102703814941082,0.00724489345550854,-0.0141742320669124,-0.999873288030067],[0,0,0,0],[8.999999E+09,8.999999E+09,8.999999E+09,8.999999E+09,8.999999E+09,8.999999E+09]];
	LOCAL CONST Robtarget Tr_meulage_motif_2_P12 :=[[-123.8128359375,-130.553046875,0.957639221191406],[-0.000102703814941082,0.00724489345550854,-0.0141742320669124,-0.999873288030067],[0,0,0,0],[8.999999E+09,8.999999E+09,8.999999E+09,8.999999E+09,8.999999E+09,8.999999E+09]];
	LOCAL CONST Robtarget Tr_meulage_motif_2_P13 :=[[-123.441140625,-131.48140625,0.959209106445313],[-0.000102703814941082,0.00724489345550854,-0.0141742320669124,-0.999873288030067],[0,0,0,0],[8.999999E+09,8.999999E+09,8.999999E+09,8.999999E+09,8.999999E+09,8.999999E+09]];
	LOCAL CONST Robtarget Tr_meulage_motif_2_P14 :=[[-123.0694453125,-132.40975,0.960778991699219],[-0.000102703814941082,0.00724489345550854,-0.0141742320669124,-0.999873288030067],[0,0,0,0],[8.999999E+09,8.999999E+09,8.999999E+09,8.999999E+09,8.999999E+09,8.999999E+09]];
	LOCAL CONST Robtarget Tr_meulage_motif_2_P15 :=[[-122.69775,-133.338109375,0.962348876953125],[-0.000102703814941082,0.00724489345550854,-0.0141742320669124,-0.999873288030067],[0,0,0,0],[8.999999E+09,8.999999E+09,8.999999E+09,8.999999E+09,8.999999E+09,8.999999E+09]];
	LOCAL CONST Robtarget Tr_meulage_motif_2_P16 :=[[-122.326046875,-134.266453125,0.963918823242187],[-0.000102703814941082,0.00724489345550854,-0.0141742320669124,-0.999873288030067],[0,0,0,0],[8.999999E+09,8.999999E+09,8.999999E+09,8.999999E+09,8.999999E+09,8.999999E+09]];
	LOCAL CONST Robtarget Tr_meulage_motif_2_P17 :=[[-121.9543515625,-135.1948125,0.965488708496094],[-0.000102703814941082,0.00724489345550854,-0.0141742320669124,-0.999873288030067],[0,0,0,0],[8.999999E+09,8.999999E+09,8.999999E+09,8.999999E+09,8.999999E+09,8.999999E+09]];
	LOCAL CONST Robtarget Tr_meulage_motif_2_P18 :=[[-121.58265625,-136.123171875,0.96705859375],[-0.000102703814941082,0.00724489345550854,-0.0141742320669124,-0.999873288030067],[0,0,0,0],[8.999999E+09,8.999999E+09,8.999999E+09,8.999999E+09,8.999999E+09,8.999999E+09]];
	LOCAL CONST Robtarget Tr_meulage_motif_2_P19 :=[[-121.1110546875,-137.0035,0.968544982910156],[-0.000102703814941082,0.00724489345550854,-0.0141742320669124,-0.999873288030067],[0,0,0,0],[8.999999E+09,8.999999E+09,8.999999E+09,8.999999E+09,8.999999E+09,8.999999E+09]];
	LOCAL CONST Robtarget Tr_meulage_motif_2_P20 :=[[-120.5631875,-137.803703125,0.969893737792969],[-0.000102703814941082,0.00724489345550854,-0.0141742320669124,-0.999873288030067],[0,0,0,0],[8.999999E+09,8.999999E+09,8.999999E+09,8.999999E+09,8.999999E+09,8.999999E+09]];
	LOCAL CONST Robtarget Tr_meulage_motif_2_P21 :=[[-119.9938671875,-138.49428125,0.971055847167969],[-0.000102703814941082,0.00724489345550854,-0.0141742320669124,-0.999873288030067],[0,0,0,0],[8.999999E+09,8.999999E+09,8.999999E+09,8.999999E+09,8.999999E+09,8.999999E+09]];
	LOCAL CONST Robtarget Tr_meulage_motif_2_P22 :=[[-119.458953125,-139.087921875,0.972053955078125],[-0.000102703814941082,0.00724489345550854,-0.0141742320669124,-0.999873288030067],[0,0,0,0],[8.999999E+09,8.999999E+09,8.999999E+09,8.999999E+09,8.999999E+09,8.999999E+09]];
	LOCAL CONST Robtarget Tr_meulage_motif_2_P23 :=[[-118.4777109375,-139.881078125,0.973382385253906],[-0.000102703814941082,0.00724489345550854,-0.0141742320669124,-0.999873288030067],[0,0,0,0],[8.999999E+09,8.999999E+09,8.999999E+09,8.999999E+09,8.999999E+09,8.999999E+09]];
	LOCAL CONST Robtarget Tr_meulage_motif_2_P24 :=[[-117.31021875,-140.51653125,0.974439208984375],[-0.000102703814941082,0.00724489345550854,-0.0141742320669124,-0.999873288030067],[0,0,0,0],[8.999999E+09,8.999999E+09,8.999999E+09,8.999999E+09,8.999999E+09,8.999999E+09]];
	LOCAL CONST Robtarget Tr_meulage_motif_2_P25 :=[[-116.044625,-140.922890625,0.97510498046875],[-0.000102703814941082,0.00724489345550854,-0.0141742320669124,-0.999873288030067],[0,0,0,0],[8.999999E+09,8.999999E+09,8.999999E+09,8.999999E+09,8.999999E+09,8.999999E+09]];
	LOCAL CONST Robtarget Tr_meulage_motif_2_P26 :=[[-114.8269609375,-140.9611875,0.975146423339844],[-0.000102703814941082,0.00724489345550854,-0.0141742320669124,-0.999873288030067],[0,0,0,0],[8.999999E+09,8.999999E+09,8.999999E+09,8.999999E+09,8.999999E+09,8.999999E+09]];
	LOCAL CONST Robtarget Tr_meulage_motif_2_P27 :=[[-114.170796875,-140.727625,0.974736938476563],[-0.000102703814941082,0.00724489345550854,-0.0141742320669124,-0.999873288030067],[0,0,0,0],[8.999999E+09,8.999999E+09,8.999999E+09,8.999999E+09,8.999999E+09,8.999999E+09]];
	LOCAL CONST Robtarget Tr_meulage_motif_2_P28 :=[[-113.556921875,-140.48184375,0.974307495117188],[-0.000102703814941082,0.00724489345550854,-0.0141742320669124,-0.999873288030067],[0,0,0,0],[8.999999E+09,8.999999E+09,8.999999E+09,8.999999E+09,8.999999E+09,8.999999E+09]];
	LOCAL CONST Robtarget Tr_meulage_motif_2_P29 :=[[-112.96359375,-140.185171875,0.9737919921875],[-0.000102703814941082,0.00724489345550854,-0.0141742320669124,-0.999873288030067],[0,0,0,0],[8.999999E+09,8.999999E+09,8.999999E+09,8.999999E+09,8.999999E+09,8.999999E+09]];
	LOCAL CONST Robtarget Tr_meulage_motif_2_P30 :=[[-112.1259609375,-139.313125,0.972294311523437],[-0.000102703814941082,0.00724489345550854,-0.0141742320669124,-0.999873288030067],[0,0,0,0],[8.999999E+09,8.999999E+09,8.999999E+09,8.999999E+09,8.999999E+09,8.999999E+09]];
	LOCAL CONST Robtarget Tr_meulage_motif_2_P31 :=[[-111.509859375,-138.14371875,0.970295776367188],[-0.000102703814941082,0.00724489345550854,-0.0141742320669124,-0.999873288030067],[0,0,0,0],[8.999999E+09,8.999999E+09,8.999999E+09,8.999999E+09,8.999999E+09,8.999999E+09]];
	LOCAL CONST Robtarget Tr_meulage_motif_2_P32 :=[[-111.120765625,-136.885546875,0.968150817871094],[-0.000102703814941082,0.00724489345550854,-0.0141742320669124,-0.999873288030067],[0,0,0,0],[8.999999E+09,8.999999E+09,8.999999E+09,8.999999E+09,8.999999E+09,8.999999E+09]];
	LOCAL CONST Robtarget Tr_meulage_motif_2_P33 :=[[-111.0087578125,-136.10059375,0.966815124511719],[-0.000102703814941082,0.00724489345550854,-0.0141742320669124,-0.999873288030067],[0,0,0,0],[8.999999E+09,8.999999E+09,8.999999E+09,8.999999E+09,8.999999E+09,8.999999E+09]];
	LOCAL CONST Robtarget Tr_meulage_motif_2_P34 :=[[-110.986640625,-134.844203125,0.964680297851563],[-0.000102703814941082,0.00724489345550854,-0.0141742320669124,-0.999873288030067],[0,0,0,0],[8.999999E+09,8.999999E+09,8.999999E+09,8.999999E+09,8.999999E+09,8.999999E+09]];
	LOCAL CONST Robtarget Tr_meulage_motif_2_P35 :=[[-111.0555625,-133.961546875,0.963182189941406],[-0.000102703814941082,0.00724489345550854,-0.0141742320669124,-0.999873288030067],[0,0,0,0],[8.999999E+09,8.999999E+09,8.999999E+09,8.999999E+09,8.999999E+09,8.999999E+09]];
	LOCAL CONST Robtarget Tr_meulage_motif_2_P36 :=[[-111.2121640625,-133.020328125,0.961586242675781],[-0.000102703814941082,0.00724489345550854,-0.0141742320669124,-0.999873288030067],[0,0,0,0],[8.999999E+09,8.999999E+09,8.999999E+09,8.999999E+09,8.999999E+09,8.999999E+09]];
	LOCAL CONST Robtarget Tr_meulage_motif_2_P37 :=[[-111.4761953125,-132.06871875,0.959974792480469],[-0.000102703814941082,0.00724489345550854,-0.0141742320669124,-0.999873288030067],[0,0,0,0],[8.999999E+09,8.999999E+09,8.999999E+09,8.999999E+09,8.999999E+09,8.999999E+09]];
	LOCAL CONST Robtarget Tr_meulage_motif_2_P38 :=[[-111.742453125,-131.106171875,0.9583447265625],[-0.000102703814941082,0.00724489345550854,-0.0141742320669124,-0.999873288030067],[0,0,0,0],[8.999999E+09,8.999999E+09,8.999999E+09,8.999999E+09,8.999999E+09,8.999999E+09]];
	LOCAL CONST Robtarget Tr_meulage_motif_2_P39 :=[[-112.1141484375,-130.1778125,0.956774841308594],[-0.000102703814941082,0.00724489345550854,-0.0141742320669124,-0.999873288030067],[0,0,0,0],[8.999999E+09,8.999999E+09,8.999999E+09,8.999999E+09,8.999999E+09,8.999999E+09]];
	LOCAL CONST Robtarget Tr_meulage_motif_2_P40 :=[[-112.48584375,-129.2494609375,0.955204956054687],[-0.000102703814941082,0.00724489345550854,-0.0141742320669124,-0.999873288030067],[0,0,0,0],[8.999999E+09,8.999999E+09,8.999999E+09,8.999999E+09,8.999999E+09,8.999999E+09]];
	LOCAL CONST Robtarget Tr_meulage_motif_2_P41 :=[[-112.8575390625,-128.3211015625,0.953635070800781],[-0.000102703814941082,0.00724489345550854,-0.0141742320669124,-0.999873288030067],[0,0,0,0],[8.999999E+09,8.999999E+09,8.999999E+09,8.999999E+09,8.999999E+09,8.999999E+09]];
	LOCAL CONST Robtarget Tr_meulage_motif_2_P42 :=[[-113.229234375,-127.39275,0.952065185546875],[-0.000102703814941082,0.00724489345550854,-0.0141742320669124,-0.999873288030067],[0,0,0,0],[8.999999E+09,8.999999E+09,8.999999E+09,8.999999E+09,8.999999E+09,8.999999E+09]];
	LOCAL CONST Robtarget Tr_meulage_motif_2_P43 :=[[-113.6009375,-126.4643984375,0.950495300292969],[-0.000102703814941082,0.00724489345550854,-0.0141742320669124,-0.999873288030067],[0,0,0,0],[8.999999E+09,8.999999E+09,8.999999E+09,8.999999E+09,8.999999E+09,8.999999E+09]];
	LOCAL CONST Robtarget Tr_meulage_motif_2_P44 :=[[-113.9726328125,-125.536046875,0.948925415039062],[-0.000102703814941082,0.00724489345550854,-0.0141742320669124,-0.999873288030067],[0,0,0,0],[8.999999E+09,8.999999E+09,8.999999E+09,8.999999E+09,8.999999E+09,8.999999E+09]];
	LOCAL CONST Robtarget Tr_meulage_motif_2_P45 :=[[-114.344328125,-124.6076953125,0.947355529785156],[-0.000102703814941082,0.00724489345550854,-0.0141742320669124,-0.999873288030067],[0,0,0,0],[8.999999E+09,8.999999E+09,8.999999E+09,8.999999E+09,8.999999E+09,8.999999E+09]];
	LOCAL CONST Robtarget Tr_meulage_motif_2_P46 :=[[-114.7160234375,-123.6793359375,0.945785583496094],[-0.000102703814941082,0.00724489345550854,-0.0141742320669124,-0.999873288030067],[0,0,0,0],[8.999999E+09,8.999999E+09,8.999999E+09,8.999999E+09,8.999999E+09,8.999999E+09]];
	LOCAL CONST Robtarget Tr_meulage_motif_2_P47 :=[[-115.08771875,-122.750984375,0.944215698242188],[-0.000102703814941082,0.00724489345550854,-0.0141742320669124,-0.999873288030067],[0,0,0,0],[8.999999E+09,8.999999E+09,8.999999E+09,8.999999E+09,8.999999E+09,8.999999E+09]];
	LOCAL CONST Robtarget Tr_meulage_motif_2_P48 :=[[-115.4594140625,-121.8226328125,0.942645812988281],[-0.000102703814941082,0.00724489345550854,-0.0141742320669124,-0.999873288030067],[0,0,0,0],[8.999999E+09,8.999999E+09,8.999999E+09,8.999999E+09,8.999999E+09,8.999999E+09]];
	LOCAL CONST Robtarget Tr_meulage_motif_2_P49 :=[[-115.725671875,-120.860078125,0.941015808105469],[-0.000102703814941082,0.00724489345550854,-0.0141742320669124,-0.999873288030067],[0,0,0,0],[8.999999E+09,8.999999E+09,8.999999E+09,8.999999E+09,8.999999E+09,8.999999E+09]];
	LOCAL CONST Robtarget Tr_meulage_motif_2_P50 :=[[-115.8814296875,-119.902890625,0.939392700195313],[-0.000102703814941082,0.00724489345550854,-0.0141742320669124,-0.999873288030067],[0,0,0,0],[8.999999E+09,8.999999E+09,8.999999E+09,8.999999E+09,8.999999E+09,8.999999E+09]];
	LOCAL CONST Robtarget Tr_meulage_motif_2_P51 :=[[-115.946015625,-119.0102265625,0.937877502441406],[-0.000102703814941082,0.00724489345550854,-0.0141742320669124,-0.999873288030067],[0,0,0,0],[8.999999E+09,8.999999E+09,8.999999E+09,8.999999E+09,8.999999E+09,8.999999E+09]];
	LOCAL CONST Robtarget Tr_meulage_motif_2_P52 :=[[-115.928109375,-118.2366484375,0.93656298828125],[-0.000102703814941082,0.00724489345550854,-0.0141742320669124,-0.999873288030067],[0,0,0,0],[8.999999E+09,8.999999E+09,8.999999E+09,8.999999E+09,8.999999E+09,8.999999E+09]];
	LOCAL CONST Robtarget Tr_meulage_motif_2_P53 :=[[-115.6975546875,-117.0300390625,0.934508728027344],[-0.000102703814941082,0.00724489345550854,-0.0141742320669124,-0.999873288030067],[0,0,0,0],[8.999999E+09,8.999999E+09,8.999999E+09,8.999999E+09,8.999999E+09,8.999999E+09]];
	LOCAL CONST Robtarget Tr_meulage_motif_2_P54 :=[[-115.195484375,-115.8574765625,0.932507019042969],[-0.000102703814941082,0.00724489345550854,-0.0141742320669124,-0.999873288030067],[0,0,0,0],[8.999999E+09,8.999999E+09,8.999999E+09,8.999999E+09,8.999999E+09,8.999999E+09]];
	LOCAL CONST Robtarget Tr_meulage_motif_2_P55 :=[[-114.4232421875,-114.97203125,0.93098779296875],[-0.000102703814941082,0.00724489345550854,-0.0141742320669124,-0.999873288030067],[0,0,0,0],[8.999999E+09,8.999999E+09,8.999999E+09,8.999999E+09,8.999999E+09,8.999999E+09]];
	LOCAL CONST Robtarget Tr_meulage_motif_2_P56 :=[[-113.8483671875,-114.5428203125,0.930247497558594],[-0.000102703814941082,0.00724489345550854,-0.0141742320669124,-0.999873288030067],[0,0,0,0],[8.999999E+09,8.999999E+09,8.999999E+09,8.999999E+09,8.999999E+09,8.999999E+09]];
	LOCAL CONST Robtarget Tr_meulage_motif_2_P57 :=[[-113.157265625,-114.19734375,0.929647216796875],[-0.000102703814941082,0.00724489345550854,-0.0141742320669124,-0.999873288030067],[0,0,0,0],[8.999999E+09,8.999999E+09,8.999999E+09,8.999999E+09,8.999999E+09,8.999999E+09]];
	LOCAL CONST Robtarget Tr_meulage_motif_2_P58 :=[[-112.417671875,-113.973328125,0.929252319335938],[-0.000102703814941082,0.00724489345550854,-0.0141742320669124,-0.999873288030067],[0,0,0,0],[8.999999E+09,8.999999E+09,8.999999E+09,8.999999E+09,8.999999E+09,8.999999E+09]];
	LOCAL CONST Robtarget Tr_meulage_motif_2_P59 :=[[-111.232859375,-113.9509296875,0.929191284179688],[-0.000102703814941082,0.00724489345550854,-0.0141742320669124,-0.999873288030067],[0,0,0,0],[8.999999E+09,8.999999E+09,8.999999E+09,8.999999E+09,8.999999E+09,8.999999E+09]];
	LOCAL CONST Robtarget Tr_meulage_motif_2_P60 :=[[-110.5351328125,-114.117859375,0.929461303710937],[-0.000102703814941082,0.00724489345550854,-0.0141742320669124,-0.999873288030067],[0,0,0,0],[8.999999E+09,8.999999E+09,8.999999E+09,8.999999E+09,8.999999E+09,8.999999E+09]];
	LOCAL CONST Robtarget Tr_meulage_motif_2_P61 :=[[-109.381828125,-114.6116875,0.93027783203125],[-0.000102703814941082,0.00724489345550854,-0.0141742320669124,-0.999873288030067],[0,0,0,0],[8.999999E+09,8.999999E+09,8.999999E+09,8.999999E+09,8.999999E+09,8.999999E+09]];
	LOCAL CONST Robtarget Tr_meulage_motif_2_P62 :=[[-108.7795,-115.0014140625,0.93092822265625],[-0.000102703814941082,0.00724489345550854,-0.0141742320669124,-0.999873288030067],[0,0,0,0],[8.999999E+09,8.999999E+09,8.999999E+09,8.999999E+09,8.999999E+09,8.999999E+09]];
	LOCAL CONST Robtarget Tr_meulage_motif_2_P63 :=[[-107.8588671875,-115.836984375,0.932329895019531],[-0.000102703814941082,0.00724489345550854,-0.0141742320669124,-0.999873288030067],[0,0,0,0],[8.999999E+09,8.999999E+09,8.999999E+09,8.999999E+09,8.999999E+09,8.999999E+09]];
	LOCAL CONST Robtarget Tr_meulage_motif_2_P64 :=[[-107.277671875,-116.49359375,0.93343408203125],[-0.000102703814941082,0.00724489345550854,-0.0141742320669124,-0.999873288030067],[0,0,0,0],[8.999999E+09,8.999999E+09,8.999999E+09,8.999999E+09,8.999999E+09,8.999999E+09]];
	LOCAL CONST Robtarget Tr_meulage_motif_2_P65 :=[[-106.7414296875,-117.2828203125,0.934764404296875],[-0.000102703814941082,0.00724489345550854,-0.0141742320669124,-0.999873288030067],[0,0,0,0],[8.999999E+09,8.999999E+09,8.999999E+09,8.999999E+09,8.999999E+09,8.999999E+09]];
	LOCAL CONST Robtarget Tr_meulage_motif_2_P66 :=[[-106.2757734375,-118.1536875,0.93623486328125],[-0.000102703814941082,0.00724489345550854,-0.0141742320669124,-0.999873288030067],[0,0,0,0],[8.999999E+09,8.999999E+09,8.999999E+09,8.999999E+09,8.999999E+09,8.999999E+09]];
	LOCAL CONST Robtarget Tr_meulage_motif_2_P67 :=[[-105.804171875,-119.03403125,0.937721252441406],[-0.000102703814941082,0.00724489345550854,-0.0141742320669124,-0.999873288030067],[0,0,0,0],[8.999999E+09,8.999999E+09,8.999999E+09,8.999999E+09,8.999999E+09,8.999999E+09]];
	LOCAL CONST Robtarget Tr_meulage_motif_2_P68 :=[[-105.4324765625,-119.9623828125,0.939291137695312],[-0.000102703814941082,0.00724489345550854,-0.0141742320669124,-0.999873288030067],[0,0,0,0],[8.999999E+09,8.999999E+09,8.999999E+09,8.999999E+09,8.999999E+09,8.999999E+09]];
	LOCAL CONST Robtarget Tr_meulage_motif_2_P69 :=[[-105.06078125,-120.8907421875,0.940861022949219],[-0.000102703814941082,0.00724489345550854,-0.0141742320669124,-0.999873288030067],[0,0,0,0],[8.999999E+09,8.999999E+09,8.999999E+09,8.999999E+09,8.999999E+09,8.999999E+09]];
	LOCAL CONST Robtarget Tr_meulage_motif_2_P70 :=[[-104.6890859375,-121.81909375,0.942430908203125],[-0.000102703814941082,0.00724489345550854,-0.0141742320669124,-0.999873288030067],[0,0,0,0],[8.999999E+09,8.999999E+09,8.999999E+09,8.999999E+09,8.999999E+09,8.999999E+09]];
	LOCAL CONST Robtarget Tr_meulage_motif_2_P71 :=[[-104.317390625,-122.7474453125,0.944000793457031],[-0.000102703814941082,0.00724489345550854,-0.0141742320669124,-0.999873288030067],[0,0,0,0],[8.999999E+09,8.999999E+09,8.999999E+09,8.999999E+09,8.999999E+09,8.999999E+09]];
	LOCAL CONST Robtarget Tr_meulage_motif_2_P72 :=[[-103.9456953125,-123.675796875,0.945570678710937],[-0.000102703814941082,0.00724489345550854,-0.0141742320669124,-0.999873288030067],[0,0,0,0],[8.999999E+09,8.999999E+09,8.999999E+09,8.999999E+09,8.999999E+09,8.999999E+09]];
	LOCAL CONST Robtarget Tr_meulage_motif_2_P73 :=[[-103.574,-124.6041484375,0.947140563964844],[-0.000102703814941082,0.00724489345550854,-0.0141742320669124,-0.999873288030067],[0,0,0,0],[8.999999E+09,8.999999E+09,8.999999E+09,8.999999E+09,8.999999E+09,8.999999E+09]];
	LOCAL CONST Robtarget Tr_meulage_motif_2_P74 :=[[-103.202296875,-125.5325078125,0.94871044921875],[-0.000102703814941082,0.00724489345550854,-0.0141742320669124,-0.999873288030067],[0,0,0,0],[8.999999E+09,8.999999E+09,8.999999E+09,8.999999E+09,8.999999E+09,8.999999E+09]];
	LOCAL CONST Robtarget Tr_meulage_motif_2_P75 :=[[-102.8306015625,-126.460859375,0.950280334472656],[-0.000102703814941082,0.00724489345550854,-0.0141742320669124,-0.999873288030067],[0,0,0,0],[8.999999E+09,8.999999E+09,8.999999E+09,8.999999E+09,8.999999E+09,8.999999E+09]];
	LOCAL CONST Robtarget Tr_meulage_motif_2_P76 :=[[-102.45890625,-127.3892109375,0.951850280761719],[-0.000102703814941082,0.00724489345550854,-0.0141742320669124,-0.999873288030067],[0,0,0,0],[8.999999E+09,8.999999E+09,8.999999E+09,8.999999E+09,8.999999E+09,8.999999E+09]];
	LOCAL CONST Robtarget Tr_meulage_motif_2_P77 :=[[-102.0872109375,-128.3175625,0.953420166015625],[-0.000102703814941082,0.00724489345550854,-0.0141742320669124,-0.999873288030067],[0,0,0,0],[8.999999E+09,8.999999E+09,8.999999E+09,8.999999E+09,8.999999E+09,8.999999E+09]];
	LOCAL CONST Robtarget Tr_meulage_motif_2_P78 :=[[-101.615609375,-129.19790625,0.954906555175781],[-0.000102703814941082,0.00724489345550854,-0.0141742320669124,-0.999873288030067],[0,0,0,0],[8.999999E+09,8.999999E+09,8.999999E+09,8.999999E+09,8.999999E+09,8.999999E+09]];
	LOCAL CONST Robtarget Tr_meulage_motif_2_P79 :=[[-101.0677421875,-129.99809375,0.956255310058594],[-0.000102703814941082,0.00724489345550854,-0.0141742320669124,-0.999873288030067],[0,0,0,0],[8.999999E+09,8.999999E+09,8.999999E+09,8.999999E+09,8.999999E+09,8.999999E+09]];
	LOCAL CONST Robtarget Tr_meulage_motif_2_P80 :=[[-100.498421875,-130.6886796875,0.957417419433594],[-0.000102703814941082,0.00724489345550854,-0.0141742320669124,-0.999873288030067],[0,0,0,0],[8.999999E+09,8.999999E+09,8.999999E+09,8.999999E+09,8.999999E+09,8.999999E+09]];
	LOCAL CONST Robtarget Tr_meulage_motif_2_P81 :=[[-99.9635078125,-131.2823125,0.95841552734375],[-0.000102703814941082,0.00724489345550854,-0.0141742320669124,-0.999873288030067],[0,0,0,0],[8.999999E+09,8.999999E+09,8.999999E+09,8.999999E+09,8.999999E+09,8.999999E+09]];
	LOCAL CONST Robtarget Tr_meulage_motif_2_P82 :=[[-98.982265625,-132.075484375,0.959743957519531],[-0.000102703814941082,0.00724489345550854,-0.0141742320669124,-0.999873288030067],[0,0,0,0],[8.999999E+09,8.999999E+09,8.999999E+09,8.999999E+09,8.999999E+09,8.999999E+09]];
	LOCAL CONST Robtarget Tr_meulage_motif_2_P83 :=[[-97.796734375,-132.631375,0.960665283203125],[-0.000102703814941082,0.00724489345550854,-0.0141742320669124,-0.999873288030067],[0,0,0,0],[8.999999E+09,8.999999E+09,8.999999E+09,8.999999E+09,8.999999E+09,8.999999E+09]];
	LOCAL CONST Robtarget Tr_meulage_motif_2_P84 :=[[-96.5621328125,-132.7931875,0.960916259765625],[-0.000102703814941082,0.00724489345550854,-0.0141742320669124,-0.999873288030067],[0,0,0,0],[8.999999E+09,8.999999E+09,8.999999E+09,8.999999E+09,8.999999E+09,8.999999E+09]];
	LOCAL CONST Robtarget Tr_meulage_motif_2_P85 :=[[-95.5853515625,-132.584484375,0.960542724609375],[-0.000102703814941082,0.00724489345550854,-0.0141742320669124,-0.999873288030067],[0,0,0,0],[8.999999E+09,8.999999E+09,8.999999E+09,8.999999E+09,8.999999E+09,8.999999E+09]];
	LOCAL CONST Robtarget Tr_meulage_motif_2_P86 :=[[-95.4442265625,-132.386375,0.960203430175781],[-0.000102703814941082,0.00724489345550854,-0.0141742320669124,-0.999873288030067],[0,0,0,0],[8.999999E+09,8.999999E+09,8.999999E+09,8.999999E+09,8.999999E+09,8.999999E+09]];
	LOCAL CONST Robtarget Tr_meulage_motif_2_P87 :=[[-94.81571875,-132.001828125,0.959538024902344],[-0.000102703814941082,0.00724489345550854,-0.0141742320669124,-0.999873288030067],[0,0,0,0],[8.999999E+09,8.999999E+09,8.999999E+09,8.999999E+09,8.999999E+09,8.999999E+09]];
	LOCAL CONST Robtarget Tr_meulage_motif_2_P88 :=[[-94.2001796875,-131.01859375,0.957855712890625],[-0.000102703814941082,0.00724489345550854,-0.0141742320669124,-0.999873288030067],[0,0,0,0],[8.999999E+09,8.999999E+09,8.999999E+09,8.999999E+09,8.999999E+09,8.999999E+09]];
	LOCAL CONST Robtarget Tr_meulage_motif_2_P89 :=[[-93.9768671875,-130.3285234375,0.956679077148437],[-0.000102703814941082,0.00724489345550854,-0.0141742320669124,-0.999873288030067],[0,0,0,0],[8.999999E+09,8.999999E+09,8.999999E+09,8.999999E+09,8.999999E+09,8.999999E+09]];
	LOCAL CONST Robtarget Tr_meulage_motif_2_P90 :=[[-93.9045625,-129.08203125,0.954560119628906],[-0.000102703814941082,0.00724489345550854,-0.0141742320669124,-0.999873288030067],[0,0,0,0],[8.999999E+09,8.999999E+09,8.999999E+09,8.999999E+09,8.999999E+09,8.999999E+09]];
	LOCAL CONST Robtarget Tr_meulage_motif_2_P91 :=[[-93.973484375,-128.1993828125,0.95306201171875],[-0.000102703814941082,0.00724489345550854,-0.0141742320669124,-0.999873288030067],[0,0,0,0],[8.999999E+09,8.999999E+09,8.999999E+09,8.999999E+09,8.999999E+09,8.999999E+09]];
	LOCAL CONST Robtarget Tr_meulage_motif_2_P92 :=[[-94.1300859375,-127.25815625,0.951466064453125],[-0.000102703814941082,0.00724489345550854,-0.0141742320669124,-0.999873288030067],[0,0,0,0],[8.999999E+09,8.999999E+09,8.999999E+09,8.999999E+09,8.999999E+09,8.999999E+09]];
	LOCAL CONST Robtarget Tr_meulage_motif_2_P93 :=[[-94.3941171875,-126.3065546875,0.949854614257812],[-0.000102703814941082,0.00724489345550854,-0.0141742320669124,-0.999873288030067],[0,0,0,0],[8.999999E+09,8.999999E+09,8.999999E+09,8.999999E+09,8.999999E+09,8.999999E+09]];
	LOCAL CONST Robtarget Tr_meulage_motif_2_P94 :=[[-94.660375,-125.344,0.948224548339844],[-0.000102703814941082,0.00724489345550854,-0.0141742320669124,-0.999873288030067],[0,0,0,0],[8.999999E+09,8.999999E+09,8.999999E+09,8.999999E+09,8.999999E+09,8.999999E+09]];
	LOCAL CONST Robtarget Tr_meulage_motif_2_P95 :=[[-95.0320703125,-124.4156484375,0.946654663085937],[-0.000102703814941082,0.00724489345550854,-0.0141742320669124,-0.999873288030067],[0,0,0,0],[8.999999E+09,8.999999E+09,8.999999E+09,8.999999E+09,8.999999E+09,8.999999E+09]];
	LOCAL CONST Robtarget Tr_meulage_motif_2_P96 :=[[-95.403765625,-123.487296875,0.945084777832031],[-0.000102703814941082,0.00724489345550854,-0.0141742320669124,-0.999873288030067],[0,0,0,0],[8.999999E+09,8.999999E+09,8.999999E+09,8.999999E+09,8.999999E+09,8.999999E+09]];
	LOCAL CONST Robtarget Tr_meulage_motif_2_P97 :=[[-95.7754609375,-122.5589453125,0.943514892578125],[-0.000102703814941082,0.00724489345550854,-0.0141742320669124,-0.999873288030067],[0,0,0,0],[8.999999E+09,8.999999E+09,8.999999E+09,8.999999E+09,8.999999E+09,8.999999E+09]];
	LOCAL CONST Robtarget Tr_meulage_motif_2_P98 :=[[-96.14715625,-121.6305859375,0.941945007324219],[-0.000102703814941082,0.00724489345550854,-0.0141742320669124,-0.999873288030067],[0,0,0,0],[8.999999E+09,8.999999E+09,8.999999E+09,8.999999E+09,8.999999E+09,8.999999E+09]];
	LOCAL CONST Robtarget Tr_meulage_motif_2_P99 :=[[-96.518859375,-120.702234375,0.940375122070312],[-0.000102703814941082,0.00724489345550854,-0.0141742320669124,-0.999873288030067],[0,0,0,0],[8.999999E+09,8.999999E+09,8.999999E+09,8.999999E+09,8.999999E+09,8.999999E+09]];
	LOCAL CONST Robtarget Tr_meulage_motif_2_P100 :=[[-96.8905546875,-119.7738828125,0.93880517578125],[-0.000102703814941082,0.00724489345550854,-0.0141742320669124,-0.999873288030067],[0,0,0,0],[8.999999E+09,8.999999E+09,8.999999E+09,8.999999E+09,8.999999E+09,8.999999E+09]];
	LOCAL CONST Robtarget Tr_meulage_motif_2_P101 :=[[-97.26225,-118.84553125,0.937235290527344],[-0.000102703814941082,0.00724489345550854,-0.0141742320669124,-0.999873288030067],[0,0,0,0],[8.999999E+09,8.999999E+09,8.999999E+09,8.999999E+09,8.999999E+09,8.999999E+09]];
	LOCAL CONST Robtarget Tr_meulage_motif_2_P102 :=[[-97.6339453125,-117.9171796875,0.935665405273438],[-0.000102703814941082,0.00724489345550854,-0.0141742320669124,-0.999873288030067],[0,0,0,0],[8.999999E+09,8.999999E+09,8.999999E+09,8.999999E+09,8.999999E+09,8.999999E+09]];
	LOCAL CONST Robtarget Tr_meulage_motif_2_P103 :=[[-98.005640625,-116.9888203125,0.934095520019531],[-0.000102703814941082,0.00724489345550854,-0.0141742320669124,-0.999873288030067],[0,0,0,0],[8.999999E+09,8.999999E+09,8.999999E+09,8.999999E+09,8.999999E+09,8.999999E+09]];
	LOCAL CONST Robtarget Tr_meulage_motif_2_P104 :=[[-98.3773359375,-116.06046875,0.932525634765625],[-0.000102703814941082,0.00724489345550854,-0.0141742320669124,-0.999873288030067],[0,0,0,0],[8.999999E+09,8.999999E+09,8.999999E+09,8.999999E+09,8.999999E+09,8.999999E+09]];
	LOCAL CONST Robtarget Tr_meulage_motif_2_P105 :=[[-98.74903125,-115.1321171875,0.930955749511719],[-0.000102703814941082,0.00724489345550854,-0.0141742320669124,-0.999873288030067],[0,0,0,0],[8.999999E+09,8.999999E+09,8.999999E+09,8.999999E+09,8.999999E+09,8.999999E+09]];
	LOCAL CONST Robtarget Tr_meulage_motif_2_P106 :=[[-99.1207265625,-114.203765625,0.929385864257813],[-0.000102703814941082,0.00724489345550854,-0.0141742320669124,-0.999873288030067],[0,0,0,0],[8.999999E+09,8.999999E+09,8.999999E+09,8.999999E+09,8.999999E+09,8.999999E+09]];
	LOCAL CONST Robtarget Tr_meulage_motif_2_P107 :=[[-99.492421875,-113.2754140625,0.927815979003906],[-0.000102703814941082,0.00724489345550854,-0.0141742320669124,-0.999873288030067],[0,0,0,0],[8.999999E+09,8.999999E+09,8.999999E+09,8.999999E+09,8.999999E+09,8.999999E+09]];
	LOCAL CONST Robtarget Tr_meulage_motif_2_P108 :=[[-99.8641171875,-112.3470546875,0.926246032714844],[-0.000102703814941082,0.00724489345550854,-0.0141742320669124,-0.999873288030067],[0,0,0,0],[8.999999E+09,8.999999E+09,8.999999E+09,8.999999E+09,8.999999E+09,8.999999E+09]];
	LOCAL CONST Robtarget Tr_meulage_motif_2_P109 :=[[-100.2358125,-111.418703125,0.924676147460938],[-0.000102703814941082,0.00724489345550854,-0.0141742320669124,-0.999873288030067],[0,0,0,0],[8.999999E+09,8.999999E+09,8.999999E+09,8.999999E+09,8.999999E+09,8.999999E+09]];
	LOCAL CONST Robtarget Tr_meulage_motif_2_P110 :=[[-100.6075078125,-110.4903515625,0.923106262207031],[-0.000102703814941082,0.00724489345550854,-0.0141742320669124,-0.999873288030067],[0,0,0,0],[8.999999E+09,8.999999E+09,8.999999E+09,8.999999E+09,8.999999E+09,8.999999E+09]];
	LOCAL CONST Robtarget Tr_meulage_motif_2_P111 :=[[-100.979203125,-109.562,0.921536376953125],[-0.000102703814941082,0.00724489345550854,-0.0141742320669124,-0.999873288030067],[0,0,0,0],[8.999999E+09,8.999999E+09,8.999999E+09,8.999999E+09,8.999999E+09,8.999999E+09]];
	LOCAL CONST Robtarget Tr_meulage_motif_2_P112 :=[[-101.3508984375,-108.633640625,0.919966491699219],[-0.000102703814941082,0.00724489345550854,-0.0141742320669124,-0.999873288030067],[0,0,0,0],[8.999999E+09,8.999999E+09,8.999999E+09,8.999999E+09,8.999999E+09,8.999999E+09]];
	LOCAL CONST Robtarget Tr_meulage_motif_2_P113 :=[[-101.7226015625,-107.7052890625,0.918396606445313],[-0.000102703814941082,0.00724489345550854,-0.0141742320669124,-0.999873288030067],[0,0,0,0],[8.999999E+09,8.999999E+09,8.999999E+09,8.999999E+09,8.999999E+09,8.999999E+09]];
	LOCAL CONST Robtarget Tr_meulage_motif_2_P114 :=[[-102.094296875,-106.7769375,0.916826721191406],[-0.000102703814941082,0.00724489345550854,-0.0141742320669124,-0.999873288030067],[0,0,0,0],[8.999999E+09,8.999999E+09,8.999999E+09,8.999999E+09,8.999999E+09,8.999999E+09]];
	LOCAL CONST Robtarget Tr_meulage_motif_2_P115 :=[[-102.4659921875,-105.8485859375,0.9152568359375],[-0.000102703814941082,0.00724489345550854,-0.0141742320669124,-0.999873288030067],[0,0,0,0],[8.999999E+09,8.999999E+09,8.999999E+09,8.999999E+09,8.999999E+09,8.999999E+09]];
	LOCAL CONST Robtarget Tr_meulage_motif_2_degg1 :=[[-102.321141793638,-106.132049539505,-9.07967521734513],[-0.000102703814941082,0.00724489345550854,-0.0141742320669124,-0.999873288030067],[0,0,0,0],[8.999999E+09,8.999999E+09,8.999999E+09,8.999999E+09,8.999999E+09,8.999999E+09]];
	LOCAL CONST Robtarget Tr_meulage_motif_2_degg2 :=[[-99.5689843102681,-111.517857977597,-198.983384229715],[-0.000102703814941082,0.00724489345550854,-0.0141742320669124,-0.999873288030067],[0,0,0,0],[8.999999E+09,8.999999E+09,8.999999E+09,8.999999E+09,8.999999E+09,8.999999E+09]];
	LOCAL CONST Robtarget Tr_meulage_bavure_App1 :=[[-63.6944152666417,-422.839199064239,31.1430737839541],[0.691444401799652,-0.720194010973759,-0.0409667062065614,0.0393313457694527],[0,0,0,0],[8.999999E+09,8.999999E+09,8.999999E+09,8.999999E+09,8.999999E+09,8.999999E+09]];
	LOCAL CONST Robtarget Tr_meulage_bavure_App2 :=[[-85.2223270133321,-234.221319328212,23.4071536891977],[0.691444401799652,-0.720194010973759,-0.0409667062065614,0.0393313457694527],[0,0,0,0],[8.999999E+09,8.999999E+09,8.999999E+09,8.999999E+09,8.999999E+09,8.999999E+09]];
	LOCAL CONST Robtarget Tr_meulage_bavure_P0 :=[[-86.355375,-224.2940625,23],[0.691444401799652,-0.720194010973759,-0.0409667062065613,0.0393313457694527],[0,0,0,0],[8.999999E+09,8.999999E+09,8.999999E+09,8.999999E+09,8.999999E+09,8.999999E+09]];
	LOCAL CONST Robtarget Tr_meulage_bavure_P1 :=[[-87.500125,-224.4294375,23],[0.691561537416635,-0.720076445199066,-0.0410066707427909,0.0393828133836296],[0,0,0,0],[8.999999E+09,8.999999E+09,8.999999E+09,8.999999E+09,8.999999E+09,8.999999E+09]];
	LOCAL CONST Robtarget Tr_meulage_bavure_P2 :=[[-87.87640625,-224.4361875,23],[0.691941017549371,-0.719699285795681,-0.0410995989792017,0.0395144178962177],[0,0,0,0],[8.999999E+09,8.999999E+09,8.999999E+09,8.999999E+09,8.999999E+09,8.999999E+09]];
	LOCAL CONST Robtarget Tr_meulage_bavure_P3 :=[[-93.49990625,-225.075984375,23],[0.692567995314119,-0.719083274200688,-0.0411799148123948,0.0396614579591333],[0,0,0,0],[8.999999E+09,8.999999E+09,8.999999E+09,8.999999E+09,8.999999E+09,8.999999E+09]];
	LOCAL CONST Robtarget Tr_meulage_bavure_P4 :=[[-96.0960390625,-225.297296875,23],[0.693431834432365,-0.718247367193583,-0.0411585090140606,0.0397364775865983],[0,0,0,0],[8.999999E+09,8.999999E+09,8.999999E+09,8.999999E+09,8.999999E+09,8.999999E+09]];
	LOCAL CONST Robtarget Tr_meulage_bavure_P5 :=[[-97.284546875,-225.427515625,23],[0.694564032771776,-0.717169422008005,-0.0409441173138942,0.03965354680097],[0,0,0,0],[8.999999E+09,8.999999E+09,8.999999E+09,8.999999E+09,8.999999E+09,8.999999E+09]];
	LOCAL CONST Robtarget Tr_meulage_bavure_P6 :=[[-100.1119375,-225.644390625,23],[0.695933144733056,-0.71588289810814,-0.0404897115251044,0.0393613708966458],[0,0,0,0],[8.999999E+09,8.999999E+09,8.999999E+09,8.999999E+09,8.999999E+09,8.999999E+09]];
	LOCAL CONST Robtarget Tr_meulage_bavure_P7 :=[[-104.9613984375,-226.140765625,23],[0.697541786456693,-0.71438029219069,-0.0398126568660629,0.0388742412095096],[0,0,0,0],[8.999999E+09,8.999999E+09,8.999999E+09,8.999999E+09,8.999999E+09,8.999999E+09]];
	LOCAL CONST Robtarget Tr_meulage_bavure_P8 :=[[-106.77725,-226.308375,23],[0.699400183889907,-0.71264182146812,-0.0389674353171027,0.0382433792200882],[0,0,0,0],[8.999999E+09,8.999999E+09,8.999999E+09,8.999999E+09,8.999999E+09,8.999999E+09]];
	LOCAL CONST Robtarget Tr_meulage_bavure_P9 :=[[-110.0874921875,-226.643359375,23],[0.701464555324831,-0.710699386356956,-0.0380209404853373,0.037526896213167],[0,0,0,0],[8.999999E+09,8.999999E+09,8.999999E+09,8.999999E+09,8.999999E+09,8.999999E+09]];
	LOCAL CONST Robtarget Tr_meulage_bavure_P10 :=[[-113.5575859375,-227.021765625,23],[0.703726326394207,-0.708552015527047,-0.0370264053400852,0.0367742320091761],[0,0,0,0],[8.999999E+09,8.999999E+09,8.999999E+09,8.999999E+09,8.999999E+09,8.999999E+09]];
	LOCAL CONST Robtarget Tr_meulage_bavure_P11 :=[[-116.4548359375,-227.2301875,23],[0.706185705407883,-0.706192626342414,-0.0360121465390592,0.036011793607438],[0,0,0,0],[8.999999E+09,8.999999E+09,8.999999E+09,8.999999E+09,8.999999E+09,8.999999E+09]];
	LOCAL CONST Robtarget Tr_meulage_bavure_P12 :=[[-117.3504296875,-227.322796875,23],[0.708830182748417,-0.703621221406747,-0.0350619426455313,0.0353215088698689],[0,0,0,0],[8.999999E+09,8.999999E+09,8.999999E+09,8.999999E+09,8.999999E+09,8.999999E+09]];
	LOCAL CONST Robtarget Tr_meulage_bavure_P13 :=[[-119.8701484375,-227.34996875,23],[0.711664608500357,-0.700805902923924,-0.0344064106058233,0.034939524098663],[0,0,0,0],[8.999999E+09,8.999999E+09,8.999999E+09,8.999999E+09,8.999999E+09,8.999999E+09]];
	LOCAL CONST Robtarget Tr_meulage_bavure_P14 :=[[-120.02590625,-227.35128125,23],[0.714629010927647,-0.697764551059063,-0.0344382494643725,0.0352705968158605],[0,0,0,0],[8.999999E+09,8.999999E+09,8.999999E+09,8.999999E+09,8.999999E+09,8.999999E+09]];
	LOCAL CONST Robtarget Tr_meulage_bavure_P15 :=[[-120.081359375,-227.343046875,23],[0.717711213798741,-0.694456998344752,-0.0355937086974086,0.0367855805812386],[0,0,0,0],[8.999999E+09,8.999999E+09,8.999999E+09,8.999999E+09,8.999999E+09,8.999999E+09]];
	LOCAL CONST Robtarget Tr_meulage_bavure_P16 :=[[-123.572390625,-227.2205625,23],[0.72090109131737,-0.690843422150928,-0.0381295127100396,0.03978847658198],[0,0,0,0],[8.999999E+09,8.999999E+09,8.999999E+09,8.999999E+09,8.999999E+09,8.999999E+09]];
	LOCAL CONST Robtarget Tr_meulage_bavure_P17 :=[[-124.4144296875,-227.007828125,23],[0.724171635350482,-0.686929669515572,-0.0418792542049999,0.0441497424711335],[0,0,0,0],[8.999999E+09,8.999999E+09,8.999999E+09,8.999999E+09,8.999999E+09,8.999999E+09]];
	LOCAL CONST Robtarget Tr_meulage_bavure_P18 :=[[-129.42459375,-228.15896875,23],[0.72756980118053,-0.682708862797118,-0.046160396682871,0.0491936057478009],[0,0,0,0],[8.999999E+09,8.999999E+09,8.999999E+09,8.999999E+09,8.999999E+09,8.999999E+09]];
	LOCAL CONST Robtarget Tr_meulage_bavure_P19 :=[[-129.723296875,-228.211296875,23],[0.731135266376711,-0.678270006588123,-0.04993578867538,0.0538278499716641],[0,0,0,0],[8.999999E+09,8.999999E+09,8.999999E+09,8.999999E+09,8.999999E+09,8.999999E+09]];
	LOCAL CONST Robtarget Tr_meulage_bavure_P20 :=[[-129.913515625,-228.228421875,23],[0.73496626310314,-0.673692852381423,-0.0521766211146837,0.0569221658007083],[0,0,0,0],[8.999999E+09,8.999999E+09,8.999999E+09,8.999999E+09,8.999999E+09,8.999999E+09]];
	LOCAL CONST Robtarget Tr_meulage_bavure_P21 :=[[-130.0992421875,-228.267765625,23],[0.739138641167566,-0.669039083923295,-0.0522439005654001,0.0577178323376254],[0,0,0,0],[8.999999E+09,8.999999E+09,8.999999E+09,8.999999E+09,8.999999E+09,8.999999E+09]];
	LOCAL CONST Robtarget Tr_meulage_bavure_P22 :=[[-133.89184375,-228.762609375,23],[0.743625715330145,-0.664355469339709,-0.0500905496024969,0.0560673050775929],[0,0,0,0],[8.999999E+09,8.999999E+09,8.999999E+09,8.999999E+09,8.999999E+09,8.999999E+09]];
	LOCAL CONST Robtarget Tr_meulage_bavure_P23 :=[[-136.1976875,-229.058875,23],[0.748374139833848,-0.659581345940635,-0.0462300686702595,0.0524535572276161],[0,0,0,0],[8.999999E+09,8.999999E+09,8.999999E+09,8.999999E+09,8.999999E+09,8.999999E+09]];
	LOCAL CONST Robtarget Tr_meulage_bavure_P24 :=[[-136.684203125,-229.0609375,23],[0.753229895970174,-0.654709725881473,-0.0414900153023872,0.0477333979847976],[0,0,0,0],[8.999999E+09,8.999999E+09,8.999999E+09,8.999999E+09,8.999999E+09,8.999999E+09]];
	LOCAL CONST Robtarget Tr_meulage_bavure_P25 :=[[-138.03153125,-229.314640625,23],[0.758066623146962,-0.64973353615337,-0.0367055171913343,0.0428255983719599],[0,0,0,0],[8.999999E+09,8.999999E+09,8.999999E+09,8.999999E+09,8.999999E+09,8.999999E+09]];
	LOCAL CONST Robtarget Tr_meulage_bavure_P26 :=[[-139.371984375,-229.441375,23],[0.76280521320189,-0.644668951027053,-0.0324683355094914,0.0384181920831934],[0,0,0,0],[8.999999E+09,8.999999E+09,8.999999E+09,8.999999E+09,8.999999E+09,8.999999E+09]];
	LOCAL CONST Robtarget Tr_meulage_bavure_P27 :=[[-140.865328125,-229.31578125,23],[0.767333470008649,-0.63964219665419,-0.0290417766236432,0.0348393638637383],[0,0,0,0],[8.999999E+09,8.999999E+09,8.999999E+09,8.999999E+09,8.999999E+09,8.999999E+09]];
	LOCAL CONST Robtarget Tr_meulage_bavure_P28 :=[[-143.39190625,-229.807625,23],[0.771605234326023,-0.634742464722592,-0.0264037209481744,0.0320968745933817],[0,0,0,0],[8.999999E+09,8.999999E+09,8.999999E+09,8.999999E+09,8.999999E+09,8.999999E+09]];
	LOCAL CONST Robtarget Tr_meulage_bavure_P29 :=[[-144.120921875,-229.863859375,23],[0.775540534176111,-0.630109097402171,-0.0244174943178212,0.0300531394714949],[0,0,0,0],[8.999999E+09,8.999999E+09,8.999999E+09,8.999999E+09,8.999999E+09,8.999999E+09]];
	LOCAL CONST Robtarget Tr_meulage_bavure_P30 :=[[-144.732828125,-229.97371875,23],[0.779055286246323,-0.625876703969777,-0.0230220614194128,0.0286565365595508],[0,0,0,0],[8.999999E+09,8.999999E+09,8.999999E+09,8.999999E+09,8.999999E+09,8.999999E+09]];
	LOCAL CONST Robtarget Tr_meulage_bavure_P31 :=[[-146.39028125,-230.049328125,23],[0.78206423161308,-0.622155822612588,-0.0224265915872018,0.0281907433473733],[0,0,0,0],[8.999999E+09,8.999999E+09,8.999999E+09,8.999999E+09,8.999999E+09,8.999999E+09]];
	LOCAL CONST Robtarget Tr_meulage_bavure_P32 :=[[-148.689984375,-230.283359375,23],[0.784443581737214,-0.619069551082826,-0.0231892909234776,0.0293839204304934],[0,0,0,0],[8.999999E+09,8.999999E+09,8.999999E+09,8.999999E+09,8.999999E+09,8.999999E+09]];
	LOCAL CONST Robtarget Tr_meulage_bavure_P33 :=[[-151.3448125,-230.487703125,23],[0.786085329360714,-0.61667222773782,-0.0260788286763673,0.0332432428562675],[0,0,0,0],[8.999999E+09,8.999999E+09,8.999999E+09,8.999999E+09,8.999999E+09,8.999999E+09]];
	LOCAL CONST Robtarget Tr_meulage_bavure_P34 :=[[-152.520015625,-230.635453125,23],[0.786836046892437,-0.615006154979267,-0.0317401587168465,0.0406082131216133],[0,0,0,0],[8.999999E+09,8.999999E+09,8.999999E+09,8.999999E+09,8.999999E+09,8.999999E+09]];
	LOCAL CONST Robtarget Tr_meulage_bavure_P35 :=[[-153.436265625,-230.33396875,23],[0.786545343857574,-0.614066333787816,-0.040207335677972,0.0515007759362932],[0,0,0,0],[8.999999E+09,8.999999E+09,8.999999E+09,8.999999E+09,8.999999E+09,8.999999E+09]];
	LOCAL CONST Robtarget Tr_meulage_bavure_P36 :=[[-154.303625,-230.3944375,23],[0.785118987808109,-0.613863614009012,-0.0506414863274143,0.0647694236620677],[0,0,0,0],[8.999999E+09,8.999999E+09,8.999999E+09,8.999999E+09,8.999999E+09,8.999999E+09]];
	LOCAL CONST Robtarget Tr_meulage_bavure_P37 :=[[-156.5379375,-230.7135,23],[0.782624373244506,-0.614503241736984,-0.0613997364266679,0.0781980093424246],[0,0,0,0],[8.999999E+09,8.999999E+09,8.999999E+09,8.999999E+09,8.999999E+09,8.999999E+09]];
	LOCAL CONST Robtarget Tr_meulage_bavure_P38 :=[[-158.895890625,-230.72159375,23],[0.779341023273098,-0.616188478912349,-0.0705500797416223,0.0892301190617614],[0,0,0,0],[8.999999E+09,8.999999E+09,8.999999E+09,8.999999E+09,8.999999E+09,8.999999E+09]];
	LOCAL CONST Robtarget Tr_meulage_bavure_P39 :=[[-160.054265625,-230.8674375,23],[0.77561870130761,-0.619159285161403,-0.076554736561081,0.0958998544857053],[0,0,0,0],[8.999999E+09,8.999999E+09,8.999999E+09,8.999999E+09,8.999999E+09,8.999999E+09]];
	LOCAL CONST Robtarget Tr_meulage_bavure_P40 :=[[-161.41184375,-230.939546875,23],[0.771702440587989,-0.623525745918465,-0.0787252042606142,0.0974337189143882],[0,0,0,0],[8.999999E+09,8.999999E+09,8.999999E+09,8.999999E+09,8.999999E+09,8.999999E+09]];
	LOCAL CONST Robtarget Tr_meulage_bavure_P41 :=[[-161.958640625,-231.196375,23],[0.767625041962976,-0.629200975910024,-0.077271450045142,0.0942711507998745],[0,0,0,0],[8.999999E+09,8.999999E+09,8.999999E+09,8.999999E+09,8.999999E+09,8.999999E+09]];
	LOCAL CONST Robtarget Tr_meulage_bavure_P42 :=[[-164.10728125,-231.71740625,23],[0.763245438698624,-0.635975099500211,-0.0729657447705512,0.0875675351458516],[0,0,0,0],[8.999999E+09,8.999999E+09,8.999999E+09,8.999999E+09,8.999999E+09,8.999999E+09]];
	LOCAL CONST Robtarget Tr_meulage_bavure_P43 :=[[-165.195015625,-231.925671875,23],[0.758471875112563,-0.643530877275866,-0.0665727613796482,0.0784633168944241],[0,0,0,0],[8.999999E+09,8.999999E+09,8.999999E+09,8.999999E+09,8.999999E+09,8.999999E+09]];
	LOCAL CONST Robtarget Tr_meulage_bavure_P44 :=[[-166.587640625,-232.2606875,23],[0.753243601574779,-0.651621293640071,-0.058568052532521,0.0677019171371414],[0,0,0,0],[8.999999E+09,8.999999E+09,8.999999E+09,8.999999E+09,8.999999E+09,8.999999E+09]];
	LOCAL CONST Robtarget Tr_meulage_bavure_P45 :=[[-167.97965625,-232.389796875,23],[0.747603152890019,-0.660024858255415,-0.0488893174944284,0.0553764111219761],[0,0,0,0],[8.999999E+09,8.999999E+09,8.999999E+09,8.999999E+09,8.999999E+09,8.999999E+09]];
	LOCAL CONST Robtarget Tr_meulage_bavure_P46 :=[[-170.014546875,-232.61046875,23],[0.741636887582964,-0.668543776864276,-0.0368192093990456,0.0408447207302585],[0,0,0,0],[8.999999E+09,8.999999E+09,8.999999E+09,8.999999E+09,8.999999E+09,8.999999E+09]];
	LOCAL CONST Robtarget Tr_meulage_bavure_P47 :=[[-174.5425,-233.26890625,23],[0.735343759059897,-0.676976383433365,-0.0211220865394894,0.0229431851615919],[0,0,0,0],[8.999999E+09,8.999999E+09,8.999999E+09,8.999999E+09,8.999999E+09,8.999999E+09]];
	LOCAL CONST Robtarget Tr_meulage_bavure_P48 :=[[-176.865703125,-233.556328125,23],[0.728643512374645,-0.684893081045964,-0.000215942039591991,0.000229736247236367],[0,0,0,0],[8.999999E+09,8.999999E+09,8.999999E+09,8.999999E+09,8.999999E+09,8.999999E+09]];
	LOCAL CONST Robtarget Tr_meulage_bavure_P49 :=[[-176.9745,-233.56259375,23],[0.721124385784761,-0.691682077534689,0.0273012731185013,-0.0284633857781776],[0,0,0,0],[8.999999E+09,8.999999E+09,8.999999E+09,8.999999E+09,8.999999E+09,8.999999E+09]];
	LOCAL CONST Robtarget Tr_meulage_bavure_P50 :=[[-177.271,-233.52315625,23],[0.712107493495985,-0.696441293893681,0.0620376714301274,-0.0634331868195909],[0,0,0,0],[8.999999E+09,8.999999E+09,8.999999E+09,8.999999E+09,8.999999E+09,8.999999E+09]];
	LOCAL CONST Robtarget Tr_meulage_bavure_P51 :=[[-179.978109375,-233.15646875,23],[0.700862760159124,-0.698126020254511,0.103265871079459,-0.103670686001076],[0,0,0,0],[8.999999E+09,8.999999E+09,8.999999E+09,8.999999E+09,8.999999E+09,8.999999E+09]];
	LOCAL CONST Robtarget Tr_meulage_bavure_P52 :=[[-181.2055625,-232.566796875,23],[0.686888497900228,-0.696018787891151,0.148861688010808,-0.146908938453292],[0,0,0,0],[8.999999E+09,8.999999E+09,8.999999E+09,8.999999E+09,8.999999E+09,8.999999E+09]];
	LOCAL CONST Robtarget Tr_meulage_bavure_P53 :=[[-182.6033125,-231.8369375,23],[0.670314561420115,-0.689982479167686,0.195907383280664,-0.190323052639176],[0,0,0,0],[8.999999E+09,8.999999E+09,8.999999E+09,8.999999E+09,8.999999E+09,8.999999E+09]];
	LOCAL CONST Robtarget Tr_meulage_bavure_P54 :=[[-184.85478125,-229.3148125,23],[0.65183569293824,-0.680613784577398,0.241563018683817,-0.231349116400556],[0,0,0,0],[8.999999E+09,8.999999E+09,8.999999E+09,8.999999E+09,8.999999E+09,8.999999E+09]];
	LOCAL CONST Robtarget Tr_meulage_bavure_P55 :=[[-185.160390625,-228.971796875,23],[0.632537794426855,-0.668991139532112,0.283614166954613,-0.268160023403523],[0,0,0,0],[8.999999E+09,8.999999E+09,8.999999E+09,8.999999E+09,8.999999E+09,8.999999E+09]];
	LOCAL CONST Robtarget Tr_meulage_bavure_P56 :=[[-186.2836875,-227.080578125,23],[0.613606452335717,-0.656357453168453,0.320655502970944,-0.299770018074936],[0,0,0,0],[8.999999E+09,8.999999E+09,8.999999E+09,8.999999E+09,8.999999E+09,8.999999E+09]];
	LOCAL CONST Robtarget Tr_meulage_bavure_P57 :=[[-187.068234375,-225.793796875,23],[0.596035646871569,-0.643932248787837,0.352024150102149,-0.325840090188867],[0,0,0,0],[8.999999E+09,8.999999E+09,8.999999E+09,8.999999E+09,8.999999E+09,8.999999E+09]];
	LOCAL CONST Robtarget Tr_meulage_bavure_P58 :=[[-187.72365625,-224.1111875,23],[0.580515751651741,-0.632582008462545,0.377731606617876,-0.346641454554393],[0,0,0,0],[8.999999E+09,8.999999E+09,8.999999E+09,8.999999E+09,8.999999E+09,8.999999E+09]];
	LOCAL CONST Robtarget Tr_meulage_bavure_P59 :=[[-188.570296875,-221.921421875,23],[0.567241961261995,-0.622689168739508,0.398439747022816,-0.362960775443492],[0,0,0,0],[8.999999E+09,8.999999E+09,8.999999E+09,8.999999E+09,8.999999E+09,8.999999E+09]];
	LOCAL CONST Robtarget Tr_meulage_bavure_P60 :=[[-188.57665625,-221.906609375,23],[0.555951804016914,-0.614138459412445,0.415258509859998,-0.375914769954176],[0,0,0,0],[8.999999E+09,8.999999E+09,8.999999E+09,8.999999E+09,8.999999E+09,8.999999E+09]];
	LOCAL CONST Robtarget Tr_meulage_bavure_P61 :=[[-188.58034375,-221.89703125,23],[0.546127663576771,-0.606458549007884,0.429428606492199,-0.386708773287595],[0,0,0,0],[8.999999E+09,8.999999E+09,8.999999E+09,8.999999E+09,8.999999E+09,8.999999E+09]];
	LOCAL CONST Robtarget Tr_meulage_bavure_P62 :=[[-188.584140625,-221.885515625,23],[0.537219253734899,-0.599195289993829,0.441972567474345,-0.396258409962319],[0,0,0,0],[8.999999E+09,8.999999E+09,8.999999E+09,8.999999E+09,8.999999E+09,8.999999E+09]];
	LOCAL CONST Robtarget Tr_meulage_bavure_P63 :=[[-189.64134375,-218.65653125,23],[0.52889771481376,-0.592073199182958,0.453463026222375,-0.405077545567865],[0,0,0,0],[8.999999E+09,8.999999E+09,8.999999E+09,8.999999E+09,8.999999E+09,8.999999E+09]];
	LOCAL CONST Robtarget Tr_meulage_bavure_P64 :=[[-189.912125,-217.440515625,23],[0.521052295685844,-0.585078842687883,0.464082732406427,-0.413297072916932],[0,0,0,0],[8.999999E+09,8.999999E+09,8.999999E+09,8.999999E+09,8.999999E+09,8.999999E+09]];
	LOCAL CONST Robtarget Tr_meulage_bavure_P65 :=[[-190.342296875,-215.3478125,23],[0.513769653380979,-0.578406130226569,0.473731125340639,-0.420792006417192],[0,0,0,0],[8.999999E+09,8.999999E+09,8.999999E+09,8.999999E+09,8.999999E+09,8.999999E+09]];
	LOCAL CONST Robtarget Tr_meulage_bavure_P66 :=[[-190.725796875,-212.964453125,23],[0.507198622203804,-0.572251879145215,0.482260160344748,-0.427437109050666],[0,0,0,0],[8.999999E+09,8.999999E+09,8.999999E+09,8.999999E+09,8.999999E+09,8.999999E+09]];
	LOCAL CONST Robtarget Tr_meulage_bavure_P67 :=[[-190.865765625,-212.0749375,23],[0.501395787148783,-0.56677326433521,0.489637438977508,-0.433157603899331],[0,0,0,0],[8.999999E+09,8.999999E+09,8.999999E+09,8.999999E+09,8.999999E+09,8.999999E+09]];
	LOCAL CONST Robtarget Tr_meulage_bavure_P68 :=[[-190.9368125,-211.261203125,23],[0.49638603032093,-0.56207505666585,0.49587740105282,-0.437924813982275],[0,0,0,0],[8.999999E+09,8.999999E+09,8.999999E+09,8.999999E+09,8.999999E+09,8.999999E+09]];
	LOCAL CONST Robtarget Tr_meulage_bavure_P69 :=[[-191.09903125,-209.78884375,23],[0.49216305232247,-0.558181277120633,0.501039135870147,-0.441779329673882],[0,0,0,0],[8.999999E+09,8.999999E+09,8.999999E+09,8.999999E+09,8.999999E+09,8.999999E+09]];
	LOCAL CONST Robtarget Tr_meulage_bavure_P70 :=[[-191.31415625,-203.657515625,23],[0.488652216205319,-0.555064114795025,0.505249898452388,-0.444798134189316],[0,0,0,0],[8.999999E+09,8.999999E+09,8.999999E+09,8.999999E+09,8.999999E+09,8.999999E+09]];
	LOCAL CONST Robtarget Tr_meulage_bavure_P71 :=[[-191.34146875,-202.041328125,23],[0.485721211575253,-0.552577958309055,0.508706563284977,-0.447157843594018],[0,0,0,0],[8.999999E+09,8.999999E+09,8.999999E+09,8.999999E+09,8.999999E+09,8.999999E+09]];
	LOCAL CONST Robtarget Tr_meulage_bavure_P72 :=[[-191.53559375,-199.877,23],[0.483139866288435,-0.550476249493592,0.511709874869607,-0.44911554449517],[0,0,0,0],[8.999999E+09,8.999999E+09,8.999999E+09,8.999999E+09,8.999999E+09,8.999999E+09]];
	LOCAL CONST Robtarget Tr_meulage_bavure_P73 :=[[-191.9845625,-194.529328125,23],[0.480623437905524,-0.548474473017048,0.514609476952776,-0.450947834693701],[0,0,0,0],[8.999999E+09,8.999999E+09,8.999999E+09,8.999999E+09,8.999999E+09,8.999999E+09]];
	LOCAL CONST Robtarget Tr_meulage_bavure_P74 :=[[-191.959390625,-193.31921875,23],[0.477950109983236,-0.546313940855303,0.517676932339683,-0.452896637344037],[0,0,0,0],[8.999999E+09,8.999999E+09,8.999999E+09,8.999999E+09,8.999999E+09,8.999999E+09]];
	LOCAL CONST Robtarget Tr_meulage_bavure_P75 :=[[-192.015140625,-190.189140625,23],[0.475010399739094,-0.543870196972642,0.521039052510915,-0.455069922916439],[0,0,0,0],[8.999999E+09,8.999999E+09,8.999999E+09,8.999999E+09,8.999999E+09,8.999999E+09]];
	LOCAL CONST Robtarget Tr_meulage_bavure_P76 :=[[-192.118234375,-186.59528125,23],[0.471813366334255,-0.5411434124921,0.524678876494241,-0.457458228722015],[0,0,0,0],[8.999999E+09,8.999999E+09,8.999999E+09,8.999999E+09,8.999999E+09,8.999999E+09]];
	LOCAL CONST Robtarget Tr_meulage_bavure_P77 :=[[-192.1558125,-180.61928125,23],[0.468451034898864,-0.538224204934254,0.528482581511395,-0.459972275429861],[0,0,0,0],[8.999999E+09,8.999999E+09,8.999999E+09,8.999999E+09,8.999999E+09,8.999999E+09]];
	LOCAL CONST Robtarget Tr_meulage_bavure_P78 :=[[-192.146453125,-179.186578125,23],[0.465021989447656,-0.535224229189708,0.532330679158493,-0.462507969493592],[0,0,0,0],[8.999999E+09,8.999999E+09,8.999999E+09,8.999999E+09,8.999999E+09,8.999999E+09]];
	LOCAL CONST Robtarget Tr_meulage_bavure_P79 :=[[-192.039453125,-173.749890625,23],[0.461597490763752,-0.532213137264297,0.536141458691755,-0.465004590639469],[0,0,0,0],[8.999999E+09,8.999999E+09,8.999999E+09,8.999999E+09,8.999999E+09,8.999999E+09]];
	LOCAL CONST Robtarget Tr_meulage_bavure_P80 :=[[-191.978125,-172.045515625,23],[0.458226484372513,-0.52923679328202,0.539861370064955,-0.467425509325028],[0,0,0,0],[8.999999E+09,8.999999E+09,8.999999E+09,8.999999E+09,8.999999E+09,8.999999E+09]];
	LOCAL CONST Robtarget Tr_meulage_bavure_P81 :=[[-191.9353125,-169.948015625,23],[0.454948940964598,-0.526324462951812,0.543449535637479,-0.469751661017911],[0,0,0,0],[8.999999E+09,8.999999E+09,8.999999E+09,8.999999E+09,8.999999E+09,8.999999E+09]];
	LOCAL CONST Robtarget Tr_meulage_bavure_P82 :=[[-191.488671875,-157.520578125,23],[0.451803646085392,-0.523525071286434,0.546865284096425,-0.471946317041055],[0,0,0,0],[8.999999E+09,8.999999E+09,8.999999E+09,8.999999E+09,8.999999E+09,8.999999E+09]];
	LOCAL CONST Robtarget Tr_meulage_bavure_P83 :=[[-191.436625,-156.502625,23],[0.448853967905007,-0.520896137616752,0.550044437939588,-0.473970933289799],[0,0,0,0],[8.999999E+09,8.999999E+09,8.999999E+09,8.999999E+09,8.999999E+09,8.999999E+09]];
	LOCAL CONST Robtarget Tr_meulage_bavure_P84 :=[[-191.130375,-153.319421875,23],[0.446154923520904,-0.518493178171879,0.552932867512075,-0.475789714508578],[0,0,0,0],[8.999999E+09,8.999999E+09,8.999999E+09,8.999999E+09,8.999999E+09,8.999999E+09]];
	LOCAL CONST Robtarget Tr_meulage_bavure_P85 :=[[-190.5631875,-146.5319375,23],[0.443734422906576,-0.516347828519392,0.555506279337838,-0.477386065493442],[0,0,0,0],[8.999999E+09,8.999999E+09,8.999999E+09,8.999999E+09,8.999999E+09,8.999999E+09]];
	LOCAL CONST Robtarget Tr_meulage_bavure_P86 :=[[-190.373859375,-143.49740625,23],[0.441590275594137,-0.514458212248085,0.557772685858642,-0.478769680808252],[0,0,0,0],[8.999999E+09,8.999999E+09,8.999999E+09,8.999999E+09,8.999999E+09,8.999999E+09]];
	LOCAL CONST Robtarget Tr_meulage_bavure_P87 :=[[-190.178234375,-141.476984375,23],[0.439698217092805,-0.5127907720524,0.559763209015476,-0.479975261670858],[0,0,0,0],[8.999999E+09,8.999999E+09,8.999999E+09,8.999999E+09,8.999999E+09,8.999999E+09]];
	LOCAL CONST Robtarget Tr_meulage_bavure_P88 :=[[-189.784984375,-136.828703125,23],[0.438022139305598,-0.51129842956668,0.561520162959641,-0.481046388605685],[0,0,0,0],[8.999999E+09,8.999999E+09,8.999999E+09,8.999999E+09,8.999999E+09,8.999999E+09]];
	LOCAL CONST Robtarget Tr_meulage_bavure_P89 :=[[-189.635,-135.669609375,23],[0.436511706304689,-0.509922988456673,0.563099276891534,-0.482032447524662],[0,0,0,0],[8.999999E+09,8.999999E+09,8.999999E+09,8.999999E+09,8.999999E+09,8.999999E+09]];
	LOCAL CONST Robtarget Tr_meulage_bavure_P90 :=[[-188.824375,-130.2146015625,23],[0.435104198272456,-0.508600804758332,0.564567621992691,-0.482983393340163],[0,0,0,0],[8.999999E+09,8.999999E+09,8.999999E+09,8.999999E+09,8.999999E+09,8.999999E+09]];
	LOCAL CONST Robtarget Tr_meulage_bavure_P91 :=[[-188.411703125,-126.2028671875,23],[0.43372674749768,-0.507246199214119,0.566002250350507,-0.483966790685142],[0,0,0,0],[8.999999E+09,8.999999E+09,8.999999E+09,8.999999E+09,8.999999E+09,8.999999E+09]];
	LOCAL CONST Robtarget Tr_meulage_bavure_P92 :=[[-188.29003125,-125.2371484375,23],[0.432305653602749,-0.505767666143696,0.567479799332065,-0.485054189855833],[0,0,0,0],[8.999999E+09,8.999999E+09,8.999999E+09,8.999999E+09,8.999999E+09,8.999999E+09]];
	LOCAL CONST Robtarget Tr_meulage_bavure_P93 :=[[-188.028796875,-122.7951953125,23],[0.43077919876384,-0.504102172554366,0.569062162397129,-0.486290588913929],[0,0,0,0],[8.999999E+09,8.999999E+09,8.999999E+09,8.999999E+09,8.999999E+09,8.999999E+09]];
	LOCAL CONST Robtarget Tr_meulage_bavure_P94 :=[[-187.1625,-115.86459375,23],[0.429112532096992,-0.502216239751764,0.570782069333733,-0.487697767735315],[0,0,0,0],[8.999999E+09,8.999999E+09,8.999999E+09,8.999999E+09,8.999999E+09,8.999999E+09]];
	LOCAL CONST Robtarget Tr_meulage_bavure_P95 :=[[-186.906765625,-114.0289140625,23],[0.427312710427844,-0.500116505919377,0.572628451763056,-0.489268826153116],[0,0,0,0],[8.999999E+09,8.999999E+09,8.999999E+09,8.999999E+09,8.999999E+09,8.999999E+09]];
	LOCAL CONST Robtarget Tr_meulage_bavure_P96 :=[[-186.823875,-113.483109375,23],[0.425401170637429,-0.497830929613364,0.574575361490604,-0.490980003165649],[0,0,0,0],[8.999999E+09,8.999999E+09,8.999999E+09,8.999999E+09,8.999999E+09,8.999999E+09]];
	LOCAL CONST Robtarget Tr_meulage_bavure_P97 :=[[-186.533015625,-111.4982109375,23],[0.423403480657147,-0.495406188521574,0.576593098748955,-0.492790624319312],[0,0,0,0],[8.999999E+09,8.999999E+09,8.999999E+09,8.999999E+09,8.999999E+09,8.999999E+09]];
	LOCAL CONST Robtarget Tr_meulage_bavure_P98 :=[[-186.286328125,-109.86053125,23],[0.421365137001314,-0.492884027379282,0.578633264729349,-0.494671913315177],[0,0,0,0],[8.999999E+09,8.999999E+09,8.999999E+09,8.999999E+09,8.999999E+09,8.999999E+09]];
	LOCAL CONST Robtarget Tr_meulage_bavure_P99 :=[[-184.30890625,-97.12115625,23],[0.41932236832459,-0.490315781898315,0.580657987351307,-0.496583816861997],[0,0,0,0],[8.999999E+09,8.999999E+09,8.999999E+09,8.999999E+09,8.999999E+09,8.999999E+09]];
	LOCAL CONST Robtarget Tr_meulage_bavure_P100 :=[[-183.1731875,-90.861453125,23],[0.41731581333145,-0.487763585002338,0.582626786664823,-0.498477907785089],[0,0,0,0],[8.999999E+09,8.999999E+09,8.999999E+09,8.999999E+09,8.999999E+09,8.999999E+09]];
	LOCAL CONST Robtarget Tr_meulage_bavure_P101 :=[[-183.11378125,-90.5538203125,23],[0.415380068391567,-0.485279108500321,0.584506883350955,-0.500315189607015],[0,0,0,0],[8.999999E+09,8.999999E+09,8.999999E+09,8.999999E+09,8.999999E+09,8.999999E+09]];
	LOCAL CONST Robtarget Tr_meulage_bavure_P102 :=[[-183.080125,-90.3695078125,23],[0.413545322426953,-0.482891405594061,0.586270585717132,-0.502078636296218],[0,0,0,0],[8.999999E+09,8.999999E+09,8.999999E+09,8.999999E+09,8.999999E+09,8.999999E+09]];
	LOCAL CONST Robtarget Tr_meulage_bavure_P103 :=[[-182.882015625,-89.3316640625,23],[0.411827642116457,-0.480614631063617,0.587904426179957,-0.503761804104279],[0,0,0,0],[8.999999E+09,8.999999E+09,8.999999E+09,8.999999E+09,8.999999E+09,8.999999E+09]];
	LOCAL CONST Robtarget Tr_meulage_bavure_P104 :=[[-181.20646875,-80.7089375,23],[0.410218380342301,-0.478460269658797,0.589419968828615,-0.505352106093806],[0,0,0,0],[8.999999E+09,8.999999E+09,8.999999E+09,8.999999E+09,8.999999E+09,8.999999E+09]];
	LOCAL CONST Robtarget Tr_meulage_bavure_P105 :=[[-180.910671875,-79.15553125,23],[0.408710083607058,-0.476430240164609,0.590827231883198,-0.506846599948981],[0,0,0,0],[8.999999E+09,8.999999E+09,8.999999E+09,8.999999E+09,8.999999E+09,8.999999E+09]];
	LOCAL CONST Robtarget Tr_meulage_bavure_P106 :=[[-177.981671875,-65.798234375,23],[0.407299786767566,-0.474504120705737,0.592130107440762,-0.508266326835215],[0,0,0,0],[8.999999E+09,8.999999E+09,8.999999E+09,8.999999E+09,8.999999E+09,8.999999E+09]];
	LOCAL CONST Robtarget Tr_meulage_bavure_P107 :=[[-177.8260625,-65.12323046875,23],[0.405951676271864,-0.472650328689735,0.593364306697084,-0.509630947705728],[0,0,0,0],[8.999999E+09,8.999999E+09,8.999999E+09,8.999999E+09,8.999999E+09,8.999999E+09]];
	LOCAL CONST Robtarget Tr_meulage_bavure_P108 :=[[-177.791859375,-64.97216796875,23],[0.404613604821418,-0.470803494406617,0.594578697839843,-0.510987350648734],[0,0,0,0],[8.999999E+09,8.999999E+09,8.999999E+09,8.999999E+09,8.999999E+09,8.999999E+09]];
	LOCAL CONST Robtarget Tr_meulage_bavure_P109 :=[[-177.730796875,-64.714796875,23],[0.403213744081189,-0.468883061533646,0.595839413398614,-0.512389251089111],[0,0,0,0],[8.999999E+09,8.999999E+09,8.999999E+09,8.999999E+09,8.999999E+09,8.999999E+09]];
	LOCAL CONST Robtarget Tr_meulage_bavure_P110 :=[[-177.548109375,-63.9358203125,23],[0.401688342312182,-0.466817830332415,0.597203485521999,-0.513882852228602],[0,0,0,0],[8.999999E+09,8.999999E+09,8.999999E+09,8.999999E+09,8.999999E+09,8.999999E+09]];
	LOCAL CONST Robtarget Tr_meulage_bavure_P111 :=[[-175.373921875,-54.97083984375,23],[0.400010133090665,-0.464565766602942,0.598691964316283,-0.515498277192582],[0,0,0,0],[8.999999E+09,8.999999E+09,8.999999E+09,8.999999E+09,8.999999E+09,8.999999E+09]];
	LOCAL CONST Robtarget Tr_meulage_bavure_P112 :=[[-174.384109375,-51.27269140625,23],[0.398182250425591,-0.462141166468631,0.600299752248432,-0.517220112864432],[0,0,0,0],[8.999999E+09,8.999999E+09,8.999999E+09,8.999999E+09,8.999999E+09,8.999999E+09]];
	LOCAL CONST Robtarget Tr_meulage_bavure_P113 :=[[-172.94053125,-45.9488515625,23],[0.396259155595451,-0.459592189056139,0.601973455984467,-0.519019902947356],[0,0,0,0],[8.999999E+09,8.999999E+09,8.999999E+09,8.999999E+09,8.999999E+09,8.999999E+09]];
	LOCAL CONST Robtarget Tr_meulage_bavure_P114 :=[[-172.2131875,-43.38656640625,23],[0.394308519469046,-0.456994235584992,0.603650733541028,-0.520848204385497],[0,0,0,0],[8.999999E+09,8.999999E+09,8.999999E+09,8.999999E+09,8.999999E+09,8.999999E+09]];
	LOCAL CONST Robtarget Tr_meulage_bavure_P115 :=[[-172.035234375,-42.760984375,23],[0.3923934019642,-0.454427902682116,0.605276776233383,-0.522649713968561],[0,0,0,0],[8.999999E+09,8.999999E+09,8.999999E+09,8.999999E+09,8.999999E+09,8.999999E+09]];
	LOCAL CONST Robtarget Tr_meulage_bavure_P116 :=[[-170.57946875,-38.1838984375,23],[0.390576232571313,-0.451947886354559,0.606795887774237,-0.524396858448181],[0,0,0,0],[8.999999E+09,8.999999E+09,8.999999E+09,8.999999E+09,8.999999E+09,8.999999E+09]];
	LOCAL CONST Robtarget Tr_meulage_bavure_P117 :=[[-169.2849375,-34.0559375,23],[0.388879501947093,-0.449585353740524,0.608191297883968,-0.526069470550804],[0,0,0,0],[8.999999E+09,8.999999E+09,8.999999E+09,8.999999E+09,8.999999E+09,8.999999E+09]];
	LOCAL CONST Robtarget Tr_meulage_bavure_P118 :=[[-168.974390625,-33.13037109375,23],[0.38730390414204,-0.44732870831298,0.609462556574374,-0.527681821450391],[0,0,0,0],[8.999999E+09,8.999999E+09,8.999999E+09,8.999999E+09,8.999999E+09,8.999999E+09]];
	LOCAL CONST Robtarget Tr_meulage_bavure_P119 :=[[-168.86915625,-32.82571484375,23],[0.385812089870429,-0.445134187654473,0.610642741415941,-0.529263666471664],[0,0,0,0],[8.999999E+09,8.999999E+09,8.999999E+09,8.999999E+09,8.999999E+09,8.999999E+09]];
	LOCAL CONST Robtarget Tr_meulage_bavure_P120 :=[[-167.68825,-29.263611328125,23],[0.384344061287666,-0.442943074298474,0.61178473154932,-0.530848865240425],[0,0,0,0],[8.999999E+09,8.999999E+09,8.999999E+09,8.999999E+09,8.999999E+09,8.999999E+09]];
	LOCAL CONST Robtarget Tr_meulage_bavure_P121 :=[[-167.1690625,-27.76254296875,23],[0.382855175236581,-0.440681448845226,0.61292117139559,-0.532493580330596],[0,0,0,0],[8.999999E+09,8.999999E+09,8.999999E+09,8.999999E+09,8.999999E+09,8.999999E+09]];
	LOCAL CONST Robtarget Tr_meulage_bavure_P122 :=[[-167.04903125,-27.413513671875,23],[0.381301547698397,-0.438312221534987,0.614089120939087,-0.534215385139863],[0,0,0,0],[8.999999E+09,8.999999E+09,8.999999E+09,8.999999E+09,8.999999E+09,8.999999E+09]];
	LOCAL CONST Robtarget Tr_meulage_bavure_P123 :=[[-165.897375,-24.163390625,23],[0.379672928230514,-0.435828105175615,0.615295554319432,-0.536016521333665],[0,0,0,0],[8.999999E+09,8.999999E+09,8.999999E+09,8.999999E+09,8.999999E+09,8.999999E+09]];
	LOCAL CONST Robtarget Tr_meulage_bavure_P124 :=[[-164.3828125,-19.499787109375,23],[0.377990713241059,-0.433243592197806,0.616518561239172,-0.537892065539768],[0,0,0,0],[8.999999E+09,8.999999E+09,8.999999E+09,8.999999E+09,8.999999E+09,8.999999E+09]];
	LOCAL CONST Robtarget Tr_meulage_bavure_P125 :=[[-163.698265625,-17.57049609375,23],[0.376290273843483,-0.430594905769898,0.617726573816181,-0.539821764045442],[0,0,0,0],[8.999999E+09,8.999999E+09,8.999999E+09,8.999999E+09,8.999999E+09,8.999999E+09]];
	LOCAL CONST Robtarget Tr_meulage_bavure_P126 :=[[-162.212765625,-13.653259765625,23],[0.374615281858369,-0.427933543635181,0.618883750655494,-0.541774100529548],[0,0,0,0],[8.999999E+09,8.999999E+09,8.999999E+09,8.999999E+09,8.999999E+09,8.999999E+09]];
	LOCAL CONST Robtarget Tr_meulage_bavure_P127 :=[[-161.5853125,-11.8774716796875,23],[0.373025151195722,-0.42532948574593,0.619943535566879,-0.543706793997784],[0,0,0,0],[8.999999E+09,8.999999E+09,8.999999E+09,8.999999E+09,8.999999E+09,8.999999E+09]];
	LOCAL CONST Robtarget Tr_meulage_bavure_P128 :=[[-159.239265625,-5.7178955078125,23],[0.371591268826863,-0.422853401520141,0.620848774096857,-0.545583842738142],[0,0,0,0],[8.999999E+09,8.999999E+09,8.999999E+09,8.999999E+09,8.999999E+09,8.999999E+09]];
	LOCAL CONST Robtarget Tr_meulage_bavure_P129 :=[[-158.1518125,-2.92898559570313,23],[0.370385018078954,-0.420565448470855,0.621541284281913,-0.547381104778336],[0,0,0,0],[8.999999E+09,8.999999E+09,8.999999E+09,8.999999E+09,8.999999E+09,8.999999E+09]];
	LOCAL CONST Robtarget Tr_meulage_bavure_P130 :=[[-157.4925625,-1.26629638671875,23],[0.369418680184547,-0.418495922838939,0.622019254118357,-0.549074720601792],[0,0,0,0],[8.999999E+09,8.999999E+09,8.999999E+09,8.999999E+09,8.999999E+09,8.999999E+09]];
	LOCAL CONST Robtarget Tr_meulage_bavure_P131 :=[[-156.282265625,1.5848388671875,23],[0.368651926583187,-0.416580980493579,0.622311606071174,-0.550712546313073],[0,0,0,0],[8.999999E+09,8.999999E+09,8.999999E+09,8.999999E+09,8.999999E+09,8.999999E+09]];
	LOCAL CONST Robtarget Tr_meulage_bavure_P132 :=[[-155.63096875,3.29946899414063,23],[0.367959365650194,-0.414673012145843,0.622512855123255,-0.552385683589369],[0,0,0,0],[8.999999E+09,8.999999E+09,8.999999E+09,8.999999E+09,8.999999E+09,8.999999E+09]];
	LOCAL CONST Robtarget Tr_meulage_bavure_P133 :=[[-153.71590625,7.906341796875,23],[0.367168916468938,-0.412576470798076,0.62275008167315,-0.554211131518409],[0,0,0,0],[8.999999E+09,8.999999E+09,8.999999E+09,8.999999E+09,8.999999E+09,8.999999E+09]];
	LOCAL CONST Robtarget Tr_meulage_bavure_P134 :=[[-152.52584375,10.5785830078125,23],[0.366123540988374,-0.41012009373187,0.62313626563285,-0.556287925362975],[0,0,0,0],[8.999999E+09,8.999999E+09,8.999999E+09,8.999999E+09,8.999999E+09,8.999999E+09]];
	LOCAL CONST Robtarget Tr_meulage_bavure_P135 :=[[-151.803453125,12.318419921875,23],[0.364754039728162,-0.407220048238421,0.623711072170317,-0.558668793890296],[0,0,0,0],[8.999999E+09,8.999999E+09,8.999999E+09,8.999999E+09,8.999999E+09,8.999999E+09]];
